//All Dump relays open  ******
IF (LCP.Section[1].Peak.DumpRelay1_close = FALSE AND
	LCP.Section[1].Peak.DumpRelay2_close = FALSE AND
	LCP.Section[1].Sust.DumpRelay1_close = FALSE AND
	LCP.Section[1].Sust.DumpRelay2_close = FALSE AND
	LCP.Section[2].Peak.DumpRelay1_close = FALSE AND
	LCP.Section[2].Peak.DumpRelay2_close = FALSE AND
	LCP.Section[2].Sust.DumpRelay1_close = FALSE AND
	LCP.Section[2].Sust.DumpRelay2_close = FALSE AND
	LCP.Section[3].Peak.DumpRelay1_close = FALSE AND
	LCP.Section[3].Peak.DumpRelay2_close = FALSE AND
	LCP.Section[3].Sust.DumpRelay1_close = FALSE AND
	LCP.Section[3].Sust.DumpRelay2_close = FALSE AND
	
	LCP.Section[4].Form.DumpRelay1_close = FALSE AND
	LCP.Section[4].Form.DumpRelay2_close = FALSE AND						
	LCP.Section[4].Form.PreFormDumpRly_close = FALSE AND
	LCP.Section[4].Form.FormTrigDumpRly1_close = FALSE AND
	LCP.Section[4].Form.PreFormTrigDumpRly1_close = FALSE) OR HMI_DB.AllDumpRelaysOpenBP = TRUE //admin bypass 
	THEN
		Permissives_DB.AllDumpRelaysOpen := TRUE;
	ELSE
		Permissives_DB.AllDumpRelaysOpen := FALSE;
END_IF;
//check for cap voltage for fully discharged
FOR i := 1 TO 3 BY 1 DO
	//peak
	FOR k := 1 TO 10 BY 1 DO
		IF LCP.Section[i].Peak.Cap[k].voltageFeedback <= 10 THEN 
			LCP.Section[i].Peak.Cap[k].CapDischaged := TRUE;
			ELSE
				LCP.Section[i].Peak.Cap[k].CapDischaged := FALSE;
		END_IF;
		//check for cap fully charged*************************
		IF LCP.Section[i].Peak.Cap[k].voltageFeedback >= Setpoints.TDKLoad[i].RequiredChargedV THEN 
			LCP.Section[i].Peak.Cap[k].CapfullyCharged := TRUE;
			ELSE
				LCP.Section[i].Peak.Cap[k].CapfullyCharged := FALSE;
		END_IF;
	END_FOR;
	//sus
	IF LCP.Section[i].Sust.Cap[1].voltageFeedback <= 10 THEN
		LCP.Section[i].Sust.Cap[1].CapDischaged := TRUE;
		ELSE
			LCP.Section[i].Sust.Cap[1].CapDischaged := FALSE;
	END_IF;
	//check fo cap fully charged
	IF LCP.Section[i].Sust.Cap[1].voltageFeedback >= Setpoints.TDKLoad[i+3].RequiredChargedV THEN
		LCP.Section[i].Sust.Cap[1].CapfullyCharged := TRUE;
		ELSE
			LCP.Section[i].Sust.Cap[1].CapfullyCharged := FALSE;
	END_IF;
	
	IF LCP.Section[i].Sust.Cap[2].voltageFeedback <= 10 THEN
		LCP.Section[i].Sust.Cap[2].CapDischaged := TRUE;
		ELSE
			LCP.Section[i].Sust.Cap[2].CapDischaged := FALSE;
	END_IF;
	//check for cap fully charged
	IF LCP.Section[i].Sust.Cap[2].voltageFeedback >= Setpoints.TDKLoad[i+3].RequiredChargedV THEN
		LCP.Section[i].Sust.Cap[2].CapfullyCharged := TRUE;
		ELSE
			LCP.Section[i].Sust.Cap[2].CapfullyCharged := FALSE;
	END_IF;
END_FOR;
// form
FOR m := 1 TO 12 BY 1 DO
	IF LCP.Section[4].Form.Cap[m].voltageFeedback <= 10 THEN
		LCP.Section[4].Form.Cap[m].CapDischaged := TRUE;
		ELSE
			LCP.Section[4].Form.Cap[m].CapDischaged := FALSE;
	END_IF;
END_FOR;

//check for cap fully charged
FOR n := 1 TO 6 BY 1 DO 
	IF LCP.Section[4].Form.Cap[n].voltageFeedback >= Setpoints.TDKLoad[7].RequiredChargedV THEN
		LCP.Section[4].Form.Cap[n].CapfullyCharged := TRUE;
		ELSE
			LCP.Section[4].Form.Cap[n].CapfullyCharged := FALSE;
	END_IF;		
END_FOR

FOR p := 7 TO 12 BY 1 DO 
	IF LCP.Section[4].Form.Cap[p].voltageFeedback >= Setpoints.TDKLoad[8].RequiredChargedV THEN
		LCP.Section[4].Form.Cap[p].CapfullyCharged := TRUE;
		ELSE
			LCP.Section[4].Form.Cap[p].CapfullyCharged := FALSE;
	END_IF;		
END_FOR

//preform
IF LCP.Section[4].PreFormCapVoltageFeedback <= 10 THEN
	LCP.Section[4].PreFormCapDischarged := TRUE;
	ELSE
		LCP.Section[4].PreFormCapDischarged := FALSE;
END_IF

//preform
IF LCP.Section[4].PreFormCapVoltageFeedback >= Setpoints.GLSLoad.RequiredChargedV THEN
	LCP.Section[4].PreFormCapFullyChaged := TRUE;
	ELSE
		LCP.Section[4].PreFormCapFullyChaged := FALSE;
END_IF


//all caps discharge condition
FOR i := 1 TO 3 BY 1 DO
	IF LCP.Section[i].Peak.Cap[1].CapDischaged = TRUE AND
		LCP.Section[i].Peak.Cap[2].CapDischaged = TRUE AND
		LCP.Section[i].Peak.Cap[3].CapDischaged = TRUE AND
		LCP.Section[i].Peak.Cap[4].CapDischaged = TRUE AND
		LCP.Section[i].Peak.Cap[5].CapDischaged = TRUE AND
		LCP.Section[i].Peak.Cap[6].CapDischaged = TRUE AND
		LCP.Section[i].Peak.Cap[7].CapDischaged = TRUE AND
		LCP.Section[i].Peak.Cap[8].CapDischaged = TRUE AND
		LCP.Section[i].Peak.Cap[9].CapDischaged = TRUE AND
		LCP.Section[i].Peak.Cap[10].CapDischaged = TRUE AND
		LCP.Section[i].Sust.Cap[1].CapDischaged = TRUE AND
		LCP.Section[i].Sust.Cap[2].CapDischaged = TRUE
		THEN
			LCP.Section[i].AllCapsDischarged := TRUE; 
		ELSE
			LCP.Section[i].AllCapsDischarged := FALSE; 
	END_IF;
	
	//all caps fully charged 
	IF LCP.Section[i].Peak.Cap[1].CapFullyCharged = TRUE AND
		LCP.Section[i].Peak.Cap[2].CapFullyCharged = TRUE AND
		LCP.Section[i].Peak.Cap[3].CapFullyCharged = TRUE AND
		LCP.Section[i].Peak.Cap[4].CapFullyCharged = TRUE AND
		LCP.Section[i].Peak.Cap[5].CapFullyCharged = TRUE AND
		LCP.Section[i].Peak.Cap[6].CapFullyCharged = TRUE AND
		LCP.Section[i].Peak.Cap[7].CapFullyCharged = TRUE AND
		LCP.Section[i].Peak.Cap[8].CapFullyCharged = TRUE AND
		LCP.Section[i].Peak.Cap[9].CapFullyCharged = TRUE AND
		LCP.Section[i].Peak.Cap[10].CapFullyCharged = TRUE AND
		LCP.Section[i].Sust.Cap[1].CapFullyCharged = TRUE AND
		LCP.Section[i].Sust.Cap[2].CapFullyCharged = TRUE
		THEN
			LCP.Section[i].AllCapsFullyCharged := TRUE;
		ELSE
			LCP.Section[i].AllCapsFullyCharged := FALSE;
	END_IF
END_FOR
//form caps 
IF LCP.Section[4].Form.Cap[1].CapDischaged = TRUE AND
	LCP.Section[4].Form.Cap[2].CapDischaged = TRUE AND
	LCP.Section[4].Form.Cap[3].CapDischaged = TRUE AND
	LCP.Section[4].Form.Cap[4].CapDischaged = TRUE AND
	LCP.Section[4].Form.Cap[5].CapDischaged = TRUE AND
	LCP.Section[4].Form.Cap[6].CapDischaged = TRUE AND
	LCP.Section[4].Form.Cap[7].CapDischaged = TRUE AND
	LCP.Section[4].Form.Cap[8].CapDischaged = TRUE AND
	LCP.Section[4].Form.Cap[9].CapDischaged = TRUE AND
	LCP.Section[4].Form.Cap[10].CapDischaged = TRUE AND
	LCP.Section[4].Form.Cap[11].CapDischaged = TRUE AND
	LCP.Section[4].Form.Cap[12].CapDischaged = TRUE AND 
	LCP.Section[4].PreFormCapDischarged = TRUE
	THEN 
		LCP.Section[4].AllCapsDischarged := TRUE;
	ELSE
		LCP.Section[4].AllCapsDischarged := FALSE;	
END_IF
//checking for caps fully charged
IF LCP.Section[4].Form.Cap[1].CapFullyCharged = TRUE AND
	LCP.Section[4].Form.Cap[2].CapFullyCharged = TRUE AND
	LCP.Section[4].Form.Cap[3].CapFullyCharged = TRUE AND
	LCP.Section[4].Form.Cap[4].CapFullyCharged = TRUE AND
	LCP.Section[4].Form.Cap[5].CapFullyCharged = TRUE AND
	LCP.Section[4].Form.Cap[6].CapFullyCharged = TRUE AND
	LCP.Section[4].Form.Cap[7].CapFullyCharged = TRUE AND
	LCP.Section[4].Form.Cap[8].CapFullyCharged = TRUE AND
	LCP.Section[4].Form.Cap[9].CapFullyCharged = TRUE AND
	LCP.Section[4].Form.Cap[10].CapFullyCharged = TRUE AND
	LCP.Section[4].Form.Cap[11].CapFullyCharged = TRUE AND
	LCP.Section[4].Form.Cap[12].CapFullyCharged = TRUE AND
	LCP.Section[4].PreFormCapFullyChaged = TRUE
	THEN
		LCP.Section[4].AllCapsFullyCharged := TRUE;
	ELSE
		LCP.Section[4].AllCapsFullyCharged := FALSE;
END_IF

//all capps fully charged
IF LCP.Section[1].AllCapsFullyCharged = TRUE AND
	LCP.Section[2].AllCapsFullyCharged = TRUE AND
	LCP.Section[3].AllCapsFullyCharged = TRUE AND
	LCP.Section[4].AllCapsFullyCharged = TRUE 
	THEN
		Permissives_DB.AllSectCapsFullyCharged := TRUE;
	ELSE
		Permissives_DB.AllSectCapsFullyCharged := FALSE;
END_IF

IF LCP.Section[1].AllCapsDischarged = TRUE AND
	LCP.Section[2].AllCapsDischarged = TRUE AND
	LCP.Section[3].AllCapsDischarged = TRUE AND
	LCP.Section[4].AllCapsDischarged = TRUE 
	THEN 
		Permissives_DB.AllSectCapsDischarged := TRUE;
	ELSE
		Permissives_DB.AllSectCapsDischarged := FALSE;
END_IF


//no loss in interlock pneumatic pressure

IF (LCP.Section[1].LossPneumaticPressure = FALSE AND
	LCP.Section[2].LossPneumaticPressure = FALSE AND
	LCP.Section[3].LossPneumaticPressure = FALSE AND
	LCP.Section[4].LossPneumaticPressure = FALSE) OR HMI_DB.InterlockPressureLossBP = TRUE 
	THEN
		Permissives_DB.NoInterlockPressureLoss := TRUE;
		ELSE
			Permissives_DB.NoInterlockPressureLoss := FALSE;
END_IF;
	
IF (Permissives_DB.NoShortingUnknowns = TRUE AND
	Trips_DB.AllDCpsuOK = TRUE AND
	Trips_DB.CageEStopCircuitBroken = FALSE AND
	Trips_DB.AnyChargerOverTemp = FALSE AND
	Trips_DB.AnyEstopPressed = FALSE AND
	Trips_DB.AnyChargerInterlockOpen = FALSE AND
	Permissives_DB.NoInterlockPressureLoss = TRUE) OR HMI_DB.SafetyOKBP = TRUE // admin bypass 
	THEN
		Permissives_DB.SafetyOK := TRUE;
		ELSE
			Permissives_DB.SafetyOK := FALSE;
END_IF;

IF i > 3 THEN
	i := 1;
END_IF;

IF j > 8 THEN
	j := 1;
END_IF;

IF k > 10 THEN
	k := 1;
END_IF;

IF m > 12 THEN
	m := 1;
END_IF;

IF n > 6 THEN
	n := 1;
END_IF;

IF p > 12 THEN
	p := 7;
END_IF;

END_PROGRAM

// ---- POUs/Trips.TcPOU
PROGRAM Trips
VAR
	bTest							: BOOL;
	//delay2s : Delay2s;
	evtLogger						: FB_TcEventLogger;
	
	ACintLockRlyFaultDelay_PT		: TIME := T#2S;
	DumpRlyFaultDelay_PT			: TIME := T#2S;
	//DumpRly2FaultDelay_PT			: TIME := T#2S;
	ChrgRlyFaultDelay_PT			: TIME := T#1S;
	
	LiftMachineGNDFaultTON			: TON;
	LiftMachineGNDFaultPT			: TIME := T#2000MS;
	
	GeneralFaultDelayPT				: TIME := T#500MS;
	
	stControl						: ST_Control;
	
	i : INT := 1;  //charger 1-8
	j : INT := 1; //section 1-3
	k : INT := 1; //section 1-4, might not need 
END_VAR


//MCP Input Trips
IF MCP_IO.MasterStopPB_Pressed = TRUE THEN
	Trips_DB.MasterStopPBPressed := TRUE;	
END_IF;

IF MCP_IO.CageEstopCircuitOK = FALSE THEN
	Trips_DB.CageEStopCircuitBroken := TRUE; 
END_IF;

IF MCP_IO.RemoteModeSelected = FALSE THEN
	Trips_DB.LocalModeSelected := TRUE; //may not be a trip
	ELSE
		Trips_DB.LocalModeSelected := FALSE;
END_IF;

IF MCP_IO.PSU1_DCOK = FALSE THEN
	Trips_DB.MCPLossDCpower := TRUE; 
END_IF;

IF (MCP_IO.LiftMachineGND = TRUE AND MCP_IO.MachineGNDrlyOpen = FALSE) OR 
	(MCP_IO.LiftMachineGND = FALSE AND MCP_IO.MachineGNDrlyOpen = TRUE)
	THEN
		//delay
		LiftMachineGNDFaultTON (IN := TRUE, PT := LiftMachineGNDFaultPT);
		IF LiftMachineGNDFaultTON.Q = TRUE THEN
			Trips_DB.MachineGNDrlyFailed := TRUE;
			LiftMachineGNDFaultTON (IN := FALSE);
		END_IF
	ELSE
		LiftMachineGNDFaultTON (IN := FALSE);
END_IF

//FOR i := 1 TO 8 BY 1 DO
FOR i := 1 TO 3 BY 1 DO	//only has 3 chargers in this version
	//check for loss inhibit

	IF (MCP_IO.Charger[i].inhibit = TRUE AND MCP_IO.Charger[i].inhibited = FALSE) OR 
		(MCP_IO.Charger[i].inhibit = FALSE AND MCP_IO.Charger[i].inhibited = TRUE)
		THEN
			MCP_IO.Charger[i].LossInhibitTON (IN := TRUE, PT := GeneralFaultDelayPT);
			IF MCP_IO.Charger[i].LossInhibitTON.Q = TRUE THEN 
				MCP_IO.Charger[i].LossInhibit := TRUE; //for alarms and not an actual trip
				MCP_IO.Charger[i].LossInhibitTON (IN := FALSE);
			END_IF
		ELSE
			MCP_IO.Charger[i].LossInhibit := FALSE;
			MCP_IO.Charger[i].LossInhibitTON (IN := FALSE);
	END_IF
	//check for loss HV on signal
	IF MCP_IO.Charger[i].HV_ON = TRUE AND MCP_IO.Charger[i].HV_isON = FALSE 
		THEN
			MCP_IO.Charger[i].LossHVON_TON (IN := TRUE, PT := GeneralFaultDelayPT);
			IF MCP_IO.Charger[i].LossHVON_TON.Q = TRUE THEN
				MCP_IO.Charger[i].LossHVON := TRUE; //for alarms and not an actual trip
				MCP_IO.Charger[i].LossHVON_TON (IN := FALSE);
			END_IF
		ELSE
			MCP_IO.Charger[i].LossHVON := FALSE;
			MCP_IO.Charger[i].LossHVON_TON (IN := FALSE);
	END_IF
	//any loss inhibit signal and hv on signal
	IF MCP_IO.Charger[i].LossInhibit = TRUE THEN 
		Trips_DB.AnyLossInhibitSignal := TRUE;
	END_IF

END_FOR;

IF ((MCP_IO.Charger[1].LossHVON = TRUE AND Recipe.PeakSupplyEN = TRUE) OR
	(MCP_IO.Charger[2].LossHVON = TRUE AND Recipe.PeakSupplyEN = TRUE) OR
	(MCP_IO.Charger[3].LossHVON = TRUE AND Recipe.PeakSupplyEN = TRUE) (*OR
	(MCP_IO.Charger[4].LossHVON = TRUE AND Recipe.SustSupplyEN = TRUE) OR
	(MCP_IO.Charger[5].LossHVON = TRUE AND Recipe.SustSupplyEN = TRUE) OR
	(MCP_IO.Charger[6].LossHVON = TRUE AND Recipe.SustSupplyEN = TRUE) OR
	(MCP_IO.Charger[7].LossHVON = TRUE AND Recipe.FormSupplyEN = TRUE) OR
	(MCP_IO.Charger[8].LossHVON = TRUE AND Recipe.FormSupplyEN = TRUE)*)) AND HMI_DB.LossHVsignalBP = FALSE 
THEN
	Trips_DB.AnyLossHVONsignal := TRUE;
END_IF


// mapping pnumatic and dc power to trips
FOR k := 1 TO 4 BY 1 DO
	Trips_DB.Section[k].LossPneumaticPressure := LCP.Section[k].LossPneumaticPressure;
	Trips_DB.Section[k].LossDCPower := NOT LCP.Section[k].PSU1_DCOK;
END_FOR;


//any charge relay fail
IF Trips_DB.Section[1].Peak.ChargeRelay1_Failed = TRUE OR
	Trips_DB.Section[1].Peak.ChargeRelay2_Failed = TRUE OR
	Trips_DB.Section[1].Sust.ChargeRelay1_Failed = TRUE OR
	Trips_DB.Section[1].Sust.ChargeRelay2_Failed = TRUE OR
	Trips_DB.Section[2].Peak.ChargeRelay1_Failed = TRUE OR
	Trips_DB.Section[2].Peak.ChargeRelay2_Failed = TRUE OR
	Trips_DB.Section[2].Sust.ChargeRelay1_Failed = TRUE OR
	Trips_DB.Section[2].Sust.ChargeRelay2_Failed = TRUE OR
	Trips_DB.Section[3].Peak.ChargeRelay1_Failed = TRUE OR
	Trips_DB.Section[3].Peak.ChargeRelay2_Failed = TRUE OR
	Trips_DB.Section[3].Sust.ChargeRelay1_Failed = TRUE OR
	Trips_DB.Section[3].Sust.ChargeRelay2_Failed = TRUE OR
	Trips_DB.Section[4].Form.ChargeRelay1_Failed = TRUE OR 
	Trips_DB.Section[4].Form.ChargeRelay2_Failed = TRUE OR 
	Trips_DB.Section[4].Form.PreFormChrgRlyFailed = TRUE OR 
	Trips_DB.Section[4].Form.FormTrigChrgRlyFailed = TRUE OR
	Trips_DB.Section[4].Form.PreFormTrigChrgRlyFailed = TRUE		
	THEN 
		Trips_DB.AnyChargeRlyFail := TRUE;
	ELSE
		Trips_DB.AnyChargeRlyFail := FALSE;
END_IF;

//any dump relay fail
IF Trips_DB.Section[1].Peak.DumpRelay1_Failed = TRUE OR
	Trips_DB.Section[1].Peak.DumpRelay2_Failed = TRUE OR
	Trips_DB.Section[1].Sust.DumpRelay1_Failed = TRUE OR
	Trips_DB.Section[1].Sust.DumpRelay2_Failed = TRUE OR
	Trips_DB.Section[2].Peak.DumpRelay1_Failed = TRUE OR
	Trips_DB.Section[2].Peak.DumpRelay2_Failed = TRUE OR
	Trips_DB.Section[2].Sust.DumpRelay1_Failed = TRUE OR
	Trips_DB.Section[2].Sust.DumpRelay2_Failed = TRUE OR
	Trips_DB.Section[3].Peak.DumpRelay1_Failed = TRUE OR
	Trips_DB.Section[3].Peak.DumpRelay2_Failed = TRUE OR
	Trips_DB.Section[3].Sust.DumpRelay1_Failed = TRUE OR
	Trips_DB.Section[3].Sust.DumpRelay2_Failed = TRUE OR
	Trips_DB.Section[4].Form.DumpRelay1_Failed = TRUE OR 
	Trips_DB.Section[4].Form.DumpRelay2_Failed = TRUE OR 
	Trips_DB.Section[4].Form.PreFormDumpRlyFailed = TRUE OR 
	Trips_DB.Section[4].Form.FormTrigDumpRly1Failed = TRUE OR
	Trips_DB.Section[4].Form.PreFormTrigDumpRly1Failed = TRUE		
	THEN 
		Trips_DB.AnyDumpRlyFail := TRUE;
	ELSE
		Trips_DB.AnyDumpRlyFail := FALSE;
END_IF;

//if relays failed, chargers faulted, loss pneumatic pressure, or loss dc power then 
//Trips_DB.Section[j].SystemTripped := TRUE;

//system trip 
//section 1-3
FOR j := 1 TO 3 BY 1 DO
	IF Trips_DB.Section[j].LossDCPower = TRUE OR 
		Trips_DB.Section[j].LossPneumaticPressure = TRUE OR
		Trips_DB.Section[j].Peak.ChargeRelay1_Failed = TRUE OR
		Trips_DB.Section[j].Peak.ChargeRelay2_Failed = TRUE OR
		Trips_DB.Section[j].Peak.DumpRelay1_Failed = TRUE OR
		Trips_DB.Section[j].Peak.DumpRelay2_Failed = TRUE OR
		Trips_DB.Section[j].Sust.ChargeRelay1_Failed = TRUE OR
		Trips_DB.Section[j].Sust.ChargeRelay2_Failed = TRUE OR
		Trips_DB.Section[j].Sust.DumpRelay1_Failed = TRUE OR
		Trips_DB.Section[j].Sust.DumpRelay2_Failed = TRUE OR
		// shorted when not supposed to ?
		LCP.Section[j].Peak.ShortContact1unknown = TRUE OR // might need to  test it.  
		LCP.Section[j].Peak.ShortContact2unknown = TRUE 
		THEN
			Trips_DB.Section[j].SystemTripped := TRUE;
	END_IF;
END_FOR;

//formation
IF Trips_DB.Section[4].LossDCPower = TRUE OR 
	Trips_DB.Section[4].LossPneumaticPressure = TRUE OR
	Trips_DB.Section[4].Form.ChargeRelay1_Failed = TRUE OR
	Trips_DB.Section[4].Form.ChargeRelay2_Failed = TRUE OR
	Trips_DB.Section[4].Form.DumpRelay1_Failed = TRUE OR
	Trips_DB.Section[4].Form.DumpRelay2_Failed = TRUE OR
	Trips_DB.Section[4].Form.PreFormChrgRlyFailed = TRUE OR
	Trips_DB.Section[4].Form.FormTrigChrgRlyFailed = TRUE OR
	Trips_DB.Section[4].Form.PreFormTrigChrgRlyFailed = TRUE OR
	Trips_DB.Section[4].Form.PreFormDumpRlyFailed = TRUE OR
	Trips_DB.Section[4].Form.FormTrigDumpRly1Failed = TRUE OR
	Trips_DB.Section[4].Form.PreFormTrigDumpRly1Failed = TRUE OR 
	LCP.Section[4].Form.ShortContact1unknown = TRUE OR //might need to remove, might be too sensitive
	LCP.Section[4].Form.ShortContact2unknown = TRUE OR 
	LCP.Section[4].Form.FormTrigShortContactUnknown = TRUE OR 
	LCP.Section[4].Form.PreFormTrigShortContactUnknown = TRUE
	THEN
		Trips_DB.Section[4].SystemTripped := TRUE;
END_IF;


//Charger faults
//FOR i := 1 TO 8 BY 1 DO
FOR i := 1 TO 3 BY 1 DO
	//OVERTEMP 
	IF MCP_IO.Charger[i].OverTemp = TRUE THEN
		Trips_DB.AnyChargerOverTemp := TRUE;  
	END_IF;
	//Load faults
	IF MCP_IO.Charger[i].LoadFaulted = TRUE THEN
		Trips_DB.AnyChargerLoadFault := TRUE;  
	END_IF;
	//Interlock Open
	IF MCP_IO.Charger[i].InterlockOpen = TRUE THEN
		Trips_DB.AnyChargerInterlockOpen := TRUE;  
	END_IF;
	
END_FOR;

//Charger summary faults
//FOR i := 1 TO 8 BY 1 DO
FOR i := 1 TO 3 BY 1 DO
	IF MCP_IO.Charger[i].SummaryFaulted = TRUE THEN
		Trips_DB.AnyChargerFaulted := TRUE;  
	END_IF;
END_FOR;

//MCP trip
IF Trips_DB.AnyChargerFaulted = TRUE OR 
	Trips_DB.MasterStopPBPressed = TRUE OR
	Trips_DB.CageEStopCircuitBroken = TRUE OR
	Trips_DB.MCPLossDCpower = TRUE 
	THEN
		Trips_DB.MCPsystemTripped := TRUE;
END_IF


//*******************E-Stop Trips
IF MCP_IO.MasterStopPB_Pressed = TRUE OR MCP_IO.CageEstopCircuitOK THEN
	Trips_DB.AnyEstopPressed := TRUE;  
END_IF;	

//*********************DC PSU
IF (MCP_IO.PSU1_DCOK = TRUE AND 
	LCP.Section[1].PSU1_DCOK = TRUE AND
	LCP.Section[2].PSU1_DCOK = TRUE AND
	LCP.Section[3].PSU1_DCOK = TRUE AND
	LCP.Section[4].PSU1_DCOK = TRUE) OR HMI_DB.AlldcPSUokBP = TRUE //admin bypass 
	THEN
		TRIPS_DB.AllDCpsuOK := TRUE;
	ELSE 
		TRIPS_DB.AllDCpsuOK := FALSE;
END_IF;

//Relay faults***************************************
//section 1 - 3
FOR j := 1 TO 3 BY 1 DO
	//Peak Charge rly1
		//fail to close
	IF LCP.Section[j].Peak.CloseChargeRelay1 = TRUE AND LCP.Section[j].Peak.ChargeRelay1_close = FALSE THEN 
		//start timer
		Trips_DB.Section[j].Peak.ChrgRly1FaultDelay_TON (IN:= TRUE, PT := ChrgRlyFaultDelay_PT);
		
		IF Trips_DB.Section[j].Peak.ChrgRly1FaultDelay_TON.Q = TRUE THEN 
			Trips_DB.Section[j].Peak.ChargeRelay1_FailtoClose := TRUE; 
			Trips_DB.Section[j].Peak.ChrgRly1FaultDelay_TON (IN:= FALSE);
		END_IF;
	ELSE
		Trips_DB.Section[j].Peak.ChrgRly1FaultDelay_TON (IN:= FALSE);
	END_IF;

		//fail to open
	IF LCP.Section[j].Peak.CloseChargeRelay1 = FALSE AND LCP.Section[j].Peak.ChargeRelay1_close = TRUE THEN 
		//start timer
		Trips_DB.Section[j].Peak.ChrgRly1FaultDelay_TON (IN:= TRUE, PT := ChrgRlyFaultDelay_PT);
		
		IF Trips_DB.Section[j].Peak.ChrgRly1FaultDelay_TON.Q = TRUE THEN 
			Trips_DB.Section[j].Peak.ChargeRelay1_FailtoOpen := TRUE; 
			Trips_DB.Section[j].Peak.ChrgRly1FaultDelay_TON (IN:= FALSE);
		END_IF;
	ELSE
		Trips_DB.Section[j].Peak.ChrgRly1FaultDelay_TON (IN:= FALSE);
	END_IF;

	//Peak Charge rly2	
		//fail to close
	IF LCP.Section[j].Peak.CloseChargeRelay2 = TRUE AND LCP.Section[j].Peak.ChargeRelay2_close = FALSE THEN 
		//start timer
		Trips_DB.Section[j].Peak.ChrgRly2FaultDelay_TON (IN:= TRUE, PT := ChrgRlyFaultDelay_PT);
		
		IF Trips_DB.Section[j].Peak.ChrgRly2FaultDelay_TON.Q = TRUE THEN 
			Trips_DB.Section[j].Peak.ChargeRelay2_FailtoClose := TRUE; 
			Trips_DB.Section[j].Peak.ChrgRly2FaultDelay_TON (IN:= FALSE);
		END_IF;
	ELSE
		Trips_DB.Section[j].Peak.ChrgRly2FaultDelay_TON (IN:= FALSE);
	END_IF;
	
		//fail to open
	IF LCP.Section[j].Peak.CloseChargeRelay2 = FALSE AND LCP.Section[j].Peak.ChargeRelay2_close = TRUE THEN 
		//start timer
		Trips_DB.Section[j].Peak.ChrgRly2FaultDelay_TON (IN:= TRUE, PT := ChrgRlyFaultDelay_PT);
		
		IF Trips_DB.Section[j].Peak.ChrgRly2FaultDelay_TON.Q = TRUE THEN 
			Trips_DB.Section[j].Peak.ChargeRelay2_FailtoOpen := TRUE; 
			Trips_DB.Section[j].Peak.ChrgRly2FaultDelay_TON (IN:= FALSE);
		END_IF;
	ELSE
		Trips_DB.Section[j].Peak.ChrgRly2FaultDelay_TON (IN:= FALSE);
	END_IF;

	//Peak dump rly1
		//fail to open
	IF LCP.Section[j].Peak.OpenDumpRelay1 = TRUE AND LCP.Section[j].Peak.DumpRelay1_close = TRUE THEN 
		//start timer
		Trips_DB.Section[j].Peak.DumpRly1FaultDelay_TON (IN := TRUE, PT := DumpRlyFaultDelay_PT);

		IF Trips_DB.Section[j].Peak.DumpRly1FaultDelay_TON.Q = TRUE THEN 
			Trips_DB.Section[j].Peak.DumpRelay1_FailtoOpen := TRUE; 
			Trips_DB.Section[j].Peak.DumpRly1FaultDelay_TON (IN:= FALSE);
		END_IF; 
	ELSE
		Trips_DB.Section[j].Peak.DumpRly1FaultDelay_TON (IN:= FALSE);
	END_IF;

		//fail to close
	IF LCP.Section[j].Peak.OpenDumpRelay1 = FALSE AND LCP.Section[j].Peak.DumpRelay1_close = FALSE THEN 
		//start timer
		Trips_DB.Section[j].Peak.DumpRly1FaultDelay_TON (IN := TRUE, PT := DumpRlyFaultDelay_PT); 
		
		IF Trips_DB.Section[j].Peak.DumpRly1FaultDelay_TON.Q = TRUE THEN 
			Trips_DB.Section[j].Peak.DumpRelay1_FailtoClose := TRUE;
			Trips_DB.Section[j].Peak.DumpRly1FaultDelay_TON (IN:= FALSE);
		END_IF;
	ELSE
		Trips_DB.Section[j].Peak.DumpRly1FaultDelay_TON (IN:= FALSE);
	END_IF;

	//Peak dump rly2
		//fail to open
	IF LCP.Section[j].Peak.OpenDumpRelay2 = TRUE AND LCP.Section[j].Peak.DumpRelay2_close = TRUE THEN 
		//start timer
		Trips_DB.Section[j].Peak.DumpRly2FaultDelay_TON (IN := TRUE, PT := DumpRlyFaultDelay_PT); 
		
		IF Trips_DB.Section[j].Peak.DumpRly2FaultDelay_TON.Q = TRUE THEN 
			Trips_DB.Section[j].Peak.DumpRelay2_FailtoOpen := TRUE; 
			Trips_DB.Section[j].Peak.DumpRly2FaultDelay_TON (IN:= FALSE);
		END_IF;
	ELSE
		Trips_DB.Section[j].Peak.DumpRly2FaultDelay_TON (IN:= FALSE);
	END_IF;

		//fail to close
	IF LCP.Section[j].Peak.OpenDumpRelay2 = FALSE AND LCP.Section[j].Peak.DumpRelay2_close = FALSE THEN 
		//start timer
		Trips_DB.Section[j].Peak.DumpRly2FaultDelay_TON (IN := TRUE, PT := DumpRlyFaultDelay_PT); 
		IF Trips_DB.Section[j].Peak.DumpRly2FaultDelay_TON.Q = TRUE THEN 
			Trips_DB.Section[j].Peak.DumpRelay2_FailtoClose := TRUE; 
			
		END_IF;
	ELSE
		Trips_DB.Section[j].Peak.DumpRly2FaultDelay_TON (IN:= FALSE);
	END_IF;
//*************************************************************************************************

//Sust Charge rly1
		//fail to close
	IF LCP.Section[j].Sust.CloseChargeRelay1 = TRUE AND LCP.Section[j].Sust.ChargeRelay1_close = FALSE THEN 
		//start timer
		Trips_DB.Section[j].Sust.ChrgRly1FaultDelay_TON (IN:= TRUE, PT := ChrgRlyFaultDelay_PT);
		
		IF Trips_DB.Section[j].Sust.ChrgRly1FaultDelay_TON.Q = TRUE THEN 
			Trips_DB.Section[j].Sust.ChargeRelay1_FailtoClose := TRUE; 
			Trips_DB.Section[j].Sust.ChrgRly1FaultDelay_TON (IN:= FALSE);
		END_IF;
	ELSE
		Trips_DB.Section[j].Sust.ChrgRly1FaultDelay_TON (IN:= FALSE);	
	END_IF;

		//fail to open
	IF LCP.Section[j].Sust.CloseChargeRelay1 = FALSE AND LCP.Section[j].Sust.ChargeRelay1_close = TRUE THEN 
		//start timer
		Trips_DB.Section[j].Sust.ChrgRly1FaultDelay_TON (IN:= TRUE, PT := ChrgRlyFaultDelay_PT);
		
		IF Trips_DB.Section[j].Sust.ChrgRly1FaultDelay_TON.Q = TRUE THEN 
			Trips_DB.Section[j].Sust.ChargeRelay1_FailtoOpen := TRUE; 
			Trips_DB.Section[j].Sust.ChrgRly1FaultDelay_TON (IN:= FALSE);
		END_IF;
	ELSE
		Trips_DB.Section[j].Sust.ChrgRly1FaultDelay_TON (IN:= FALSE);
	END_IF;

	//Sust Charge rly2	
		//fail to close
	IF LCP.Section[j].Sust.CloseChargeRelay2 = TRUE AND LCP.Section[j].Sust.ChargeRelay2_close = FALSE THEN 
		//start timer
		Trips_DB.Section[j].Sust.ChrgRly2FaultDelay_TON (IN:= TRUE, PT := ChrgRlyFaultDelay_PT);
		
		IF Trips_DB.Section[j].Sust.ChrgRly2FaultDelay_TON.Q = TRUE THEN 
			Trips_DB.Section[j].Sust.ChargeRelay2_FailtoClose := TRUE;
			Trips_DB.Section[j].Sust.ChrgRly2FaultDelay_TON (IN:= FALSE);
		END_IF;
	ELSE
		Trips_DB.Section[j].Sust.ChrgRly2FaultDelay_TON (IN:= FALSE);
	END_IF;
	
		//fail to open
	IF LCP.Section[j].Sust.CloseChargeRelay2 = FALSE AND LCP.Section[j].Sust.ChargeRelay2_close = TRUE THEN 
		//start timer
		Trips_DB.Section[j].Sust.ChrgRly2FaultDelay_TON (IN:= TRUE, PT := ChrgRlyFaultDelay_PT);
		
		IF Trips_DB.Section[j].Sust.ChrgRly2FaultDelay_TON.Q = TRUE THEN 
			Trips_DB.Section[j].Sust.ChargeRelay2_FailtoOpen := TRUE; 
			Trips_DB.Section[j].Sust.ChrgRly2FaultDelay_TON (IN:= FALSE);
		END_IF;
	ELSE
		Trips_DB.Section[j].Sust.ChrgRly2FaultDelay_TON (IN:= FALSE);
	END_IF;

	//Sust dump rly1
		//fail to open
	IF LCP.Section[j].Sust.OpenDumpRelay1 = TRUE AND LCP.Section[j].Sust.DumpRelay1_close = TRUE THEN 
		//start timer
		Trips_DB.Section[j].Sust.DumpRly1FaultDelay_TON (IN := TRUE, PT := DumpRlyFaultDelay_PT);

		IF Trips_DB.Section[j].Sust.DumpRly1FaultDelay_TON.Q = TRUE THEN 
			Trips_DB.Section[j].Sust.DumpRelay1_FailtoOpen := TRUE; 
			Trips_DB.Section[j].Sust.DumpRly1FaultDelay_TON (IN:= FALSE);
		END_IF; 
	ELSE
		Trips_DB.Section[j].Sust.DumpRly1FaultDelay_TON (IN:= FALSE);
	END_IF;

		//fail to close
	IF LCP.Section[j].Sust.OpenDumpRelay1 = FALSE AND LCP.Section[j].Sust.DumpRelay1_close = FALSE THEN 
		//start timer
		Trips_DB.Section[j].Sust.DumpRly1FaultDelay_TON (IN := TRUE, PT := DumpRlyFaultDelay_PT); 
		
		IF Trips_DB.Section[j].Sust.DumpRly1FaultDelay_TON.Q = TRUE THEN 
			Trips_DB.Section[j].Sust.DumpRelay1_FailtoClose := TRUE; 
			Trips_DB.Section[j].Sust.DumpRly1FaultDelay_TON (IN:= FALSE);
		END_IF;
	ELSE
		Trips_DB.Section[j].Sust.DumpRly1FaultDelay_TON (IN:= FALSE);
	END_IF;

	//Sust dump rly2
		//fail to open
	IF LCP.Section[j].Sust.OpenDumpRelay2 = TRUE AND LCP.Section[j].Sust.DumpRelay2_close = TRUE THEN 
		//start timer
		Trips_DB.Section[j].Sust.DumpRly2FaultDelay_TON (IN := TRUE, PT := DumpRlyFaultDelay_PT); 
		
		IF Trips_DB.Section[j].Sust.DumpRly2FaultDelay_TON.Q = TRUE THEN 
			Trips_DB.Section[j].Sust.DumpRelay2_FailtoOpen := TRUE; 
			Trips_DB.Section[j].Sust.DumpRly2FaultDelay_TON (IN:= FALSE);
		END_IF;
	ELSE
		Trips_DB.Section[j].Sust.DumpRly2FaultDelay_TON (IN:= FALSE);
	END_IF;

		//fail to close
	IF LCP.Section[j].Sust.OpenDumpRelay2 = FALSE AND LCP.Section[j].Sust.DumpRelay2_close = FALSE THEN 
		//start timer
		Trips_DB.Section[j].Sust.DumpRly2FaultDelay_TON (IN := TRUE, PT := DumpRlyFaultDelay_PT); 
		IF Trips_DB.Section[j].Sust.DumpRly2FaultDelay_TON.Q = TRUE THEN 
			Trips_DB.Section[j].Sust.DumpRelay2_FailtoClose := TRUE; 
			Trips_DB.Section[j].Sust.DumpRly2FaultDelay_TON (IN:= FALSE);
		END_IF;
	ELSE
		Trips_DB.Section[j].Sust.DumpRly2FaultDelay_TON (IN:= FALSE);
	END_IF;
	
END_FOR;
//****************************************	
	
//Form Charge rly1
		//fail to close
IF LCP.Section[4].Form.CloseChargeRelay1 = TRUE AND LCP.Section[4].Form.ChargeRelay1_close = FALSE THEN 
		//start timer
		Trips_DB.Section[4].Form.ChrgRly1FaultDelay_TON (IN:= TRUE, PT := ChrgRlyFaultDelay_PT);
		
		IF Trips_DB.Section[4].Form.ChrgRly1FaultDelay_TON.Q = TRUE THEN 
			Trips_DB.Section[4].Form.ChargeRelay1_FailtoClose := TRUE; 
			Trips_DB.Section[4].Form.ChrgRly1FaultDelay_TON (IN:= FALSE);
		END_IF;
	ELSE
		Trips_DB.Section[4].Form.ChrgRly1FaultDelay_TON (IN:= FALSE);		
END_IF;

		//fail to open
IF LCP.Section[4].Form.CloseChargeRelay1 = FALSE AND LCP.Section[4].Form.ChargeRelay1_close = TRUE THEN 
		//start timer
		Trips_DB.Section[4].Form.ChrgRly1FaultDelay_TON (IN:= TRUE, PT := ChrgRlyFaultDelay_PT);
		
		IF Trips_DB.Section[4].Form.ChrgRly1FaultDelay_TON.Q = TRUE THEN 
			Trips_DB.Section[4].Form.ChargeRelay1_FailtoOpen := TRUE; 
			Trips_DB.Section[4].Form.ChrgRly1FaultDelay_TON (IN:= FALSE);
		END_IF;
	ELSE
		Trips_DB.Section[4].Form.ChrgRly1FaultDelay_TON (IN:= FALSE);
END_IF;

	//Form Charge rly2	
		//fail to close
IF LCP.Section[4].Form.CloseChargeRelay2 = TRUE AND LCP.Section[4].Form.ChargeRelay2_close = FALSE THEN 
		//start timer
		Trips_DB.Section[4].Form.ChrgRly2FaultDelay_TON (IN:= TRUE, PT := ChrgRlyFaultDelay_PT);
		
		IF Trips_DB.Section[4].Form.ChrgRly2FaultDelay_TON.Q = TRUE THEN 
			Trips_DB.Section[4].Form.ChargeRelay2_FailtoClose := TRUE; 
			Trips_DB.Section[4].Form.ChrgRly2FaultDelay_TON (IN:= FALSE);
		END_IF;
	ELSE
		Trips_DB.Section[4].Form.ChrgRly2FaultDelay_TON (IN:= FALSE);
END_IF;
	
		//fail to open
IF LCP.Section[4].Form.CloseChargeRelay2 = FALSE AND LCP.Section[4].Form.ChargeRelay2_close = TRUE THEN 
		//start timer
		Trips_DB.Section[4].Form.ChrgRly2FaultDelay_TON (IN:= TRUE, PT := ChrgRlyFaultDelay_PT);
		
		IF Trips_DB.Section[4].Form.ChrgRly2FaultDelay_TON.Q = TRUE THEN 
			Trips_DB.Section[4].Form.ChargeRelay2_FailtoOpen := TRUE; 
			Trips_DB.Section[4].Form.ChrgRly2FaultDelay_TON (IN:= FALSE);
		END_IF;
	ELSE
		Trips_DB.Section[4].Form.ChrgRly2FaultDelay_TON (IN:= FALSE);
END_IF;

	//Form dump rly1
		//fail to open
IF LCP.Section[4].Form.OpenDumpRelay1 = TRUE AND LCP.Section[4].Form.DumpRelay1_close = TRUE THEN 
		//start timer
		Trips_DB.Section[4].Form.DumpRly1FaultDelay_TON (IN := TRUE, PT := DumpRlyFaultDelay_PT);

		IF Trips_DB.Section[4].Form.DumpRly1FaultDelay_TON.Q = TRUE THEN 
			Trips_DB.Section[4].Form.DumpRelay1_FailtoOpen := TRUE; 
			Trips_DB.Section[4].Form.DumpRly1FaultDelay_TON (IN:= FALSE);
		END_IF; 
	ELSE
		Trips_DB.Section[4].Form.DumpRly1FaultDelay_TON (IN:= FALSE);
END_IF;

		//fail to close
IF LCP.Section[4].Form.OpenDumpRelay1 = FALSE AND LCP.Section[4].Form.DumpRelay1_close = FALSE THEN 
		//start timer
		Trips_DB.Section[4].Form.DumpRly1FaultDelay_TON (IN := TRUE, PT := DumpRlyFaultDelay_PT); 
		
		IF Trips_DB.Section[4].Form.DumpRly1FaultDelay_TON.Q = TRUE THEN 
			Trips_DB.Section[4].Form.DumpRelay1_FailtoClose := TRUE; 
			Trips_DB.Section[4].Form.DumpRly1FaultDelay_TON (IN:= FALSE);
		END_IF;
	ELSE
		Trips_DB.Section[4].Form.DumpRly1FaultDelay_TON (IN:= FALSE);
END_IF;

	//Form dump rly2
		//fail to open
IF LCP.Section[4].Form.OpenDumpRelay2 = TRUE AND LCP.Section[4].Form.DumpRelay2_close = TRUE THEN 
		//start timer
		Trips_DB.Section[4].Form.DumpRly2FaultDelay_TON (IN := TRUE, PT := DumpRlyFaultDelay_PT); 
		
		IF Trips_DB.Section[4].Form.DumpRly2FaultDelay_TON.Q = TRUE THEN 
			Trips_DB.Section[4].Form.DumpRelay2_FailtoOpen := TRUE; 
			Trips_DB.Section[4].Form.DumpRly2FaultDelay_TON (IN:= FALSE);
		END_IF;
	ELSE
		Trips_DB.Section[4].Form.DumpRly2FaultDelay_TON (IN:= FALSE);
END_IF;

		//fail to close
IF LCP.Section[4].Form.OpenDumpRelay2 = FALSE AND LCP.Section[4].Form.DumpRelay2_close = FALSE THEN 
		//start timer
		Trips_DB.Section[4].Form.DumpRly2FaultDelay_TON (IN := TRUE, PT := DumpRlyFaultDelay_PT); 
		IF Trips_DB.Section[4].Form.DumpRly2FaultDelay_TON.Q = TRUE THEN 
			Trips_DB.Section[4].Form.DumpRelay2_FailtoClose := TRUE; 
			Trips_DB.Section[4].Form.DumpRly2FaultDelay_TON (IN:= FALSE);
		END_IF;
	ELSE
		Trips_DB.Section[4].Form.DumpRly2FaultDelay_TON (IN:= FALSE);
END_IF;	

	//PreForm Charge rly
		//fail to close
IF (LCP.Section[4].Form.ClosePreFormChargeRly = TRUE AND LCP.Section[4].Form.PreFormChargeRly_close = FALSE) OR 
		(LCP.Section[4].Form.ClosePreFormChargeRly = FALSE AND LCP.Section[4].Form.PreFormChargeRly_close = TRUE) 
		THEN 
		//start timer
		Trips_DB.Section[4].Form.PreFormChrgRlyFaultDelay_TON (IN:= TRUE, PT := ChrgRlyFaultDelay_PT);
		
		IF Trips_DB.Section[4].Form.PreFormChrgRlyFaultDelay_TON.Q = TRUE THEN 
			Trips_DB.Section[4].Form.PreFormChrgRlyFailed := TRUE; 
			Trips_DB.Section[4].Form.PreFormChrgRlyFaultDelay_TON (IN:= FALSE);
		END_IF;
	ELSE
		Trips_DB.Section[4].Form.PreFormChrgRlyFaultDelay_TON (IN:= FALSE);
END_IF;

//form trigger charge 
		//fail to close
IF (LCP.Section[4].Form.CloseFormTrigChargeRly = TRUE AND LCP.Section[4].Form.FormTrigChargeRly_close = FALSE) OR 
		(LCP.Section[4].Form.CloseFormTrigChargeRly = FALSE AND LCP.Section[4].Form.FormTrigChargeRly_close = TRUE) 
		THEN 
		//start timer
		Trips_DB.Section[4].Form.FormTrigChrgRlyFaultDelay_TON (IN:= TRUE, PT := ChrgRlyFaultDelay_PT);
		
		IF Trips_DB.Section[4].Form.FormTrigChrgRlyFaultDelay_TON.Q = TRUE THEN 
			Trips_DB.Section[4].Form.FormTrigChrgRlyFailed := TRUE; 
			Trips_DB.Section[4].Form.FormTrigChrgRlyFaultDelay_TON (IN:= FALSE);
		END_IF;
	ELSE
		Trips_DB.Section[4].Form.FormTrigChrgRlyFaultDelay_TON (IN:= FALSE);
END_IF;

//preform trigger charge
		//fail to close
IF (LCP.Section[4].Form.ClosePreFormTrigChargeRly = TRUE AND LCP.Section[4].Form.PreFormTrigChargeRly_close = FALSE) OR 
		(LCP.Section[4].Form.ClosePreFormTrigChargeRly = FALSE AND LCP.Section[4].Form.PreFormTrigChargeRly_close = TRUE) 
		THEN 
		//start timer
		Trips_DB.Section[4].Form.PreFormTrigChrgRlyFaultDelay_TON (IN:= TRUE, PT := ChrgRlyFaultDelay_PT);
		
		IF Trips_DB.Section[4].Form.PreFormTrigChrgRlyFaultDelay_TON.Q = TRUE THEN 
			Trips_DB.Section[4].Form.PreFormTrigChrgRlyFailed := TRUE; 
			Trips_DB.Section[4].Form.PreFormTrigChrgRlyFaultDelay_TON (IN:= FALSE);
		END_IF;
	ELSE
		Trips_DB.Section[4].Form.PreFormTrigChrgRlyFaultDelay_TON (IN:= FALSE);
END_IF;

//preform dump
	//fail to close
IF (LCP.Section[4].Form.OpenPreFormDumpRly = TRUE AND LCP.Section[4].Form.PreFormDumpRly_close = FALSE) OR 
		(LCP.Section[4].Form.OpenPreFormDumpRly = FALSE AND LCP.Section[4].Form.PreFormDumpRly_close = TRUE) 
		THEN 
		//start timer
		Trips_DB.Section[4].Form.PreFormDumpRlyFaultDelay_TON (IN:= TRUE, PT := DumpRlyFaultDelay_PT);
		
		IF Trips_DB.Section[4].Form.PreFormDumpRlyFaultDelay_TON.Q = TRUE THEN 
			Trips_DB.Section[4].Form.PreFormDumpRlyFailed := TRUE; 
			Trips_DB.Section[4].Form.PreFormDumpRlyFaultDelay_TON (IN:= FALSE);
		END_IF;
	ELSE
		Trips_DB.Section[4].Form.PreFormDumpRlyFaultDelay_TON (IN:= FALSE);
END_IF;

//form trigger dump
	//fail to close
IF (LCP.Section[4].Form.OpenFormTrigDumpRly1 = TRUE AND LCP.Section[4].Form.FormTrigDumpRly1_close = FALSE) OR 
		(LCP.Section[4].Form.OpenFormTrigDumpRly1 = FALSE AND LCP.Section[4].Form.FormTrigDumpRly1_close = TRUE) 
		THEN 
		//start timer
		Trips_DB.Section[4].Form.FormTrigDumpRlyFaultDelay_TON (IN:= TRUE, PT := DumpRlyFaultDelay_PT);
		
		IF Trips_DB.Section[4].Form.FormTrigDumpRlyFaultDelay_TON.Q = TRUE THEN 
			Trips_DB.Section[4].Form.FormTrigDumpRly1Failed := TRUE; 
			Trips_DB.Section[4].Form.FormTrigDumpRlyFaultDelay_TON (IN:= FALSE);
		END_IF;
	ELSE
		Trips_DB.Section[4].Form.FormTrigDumpRlyFaultDelay_TON (IN:= FALSE);
END_IF;
	
//preform trigger dump
	//fail to close
IF (LCP.Section[4].Form.OpenPreFormTrigDumpRly1 = TRUE AND LCP.Section[4].Form.PreFormTrigDumpRly1_close = FALSE) OR 
		(LCP.Section[4].Form.OpenPreFormTrigDumpRly1 = FALSE AND LCP.Section[4].Form.PreFormTrigDumpRly1_close = TRUE) 
		THEN 
		//start timer
		Trips_DB.Section[4].Form.PreFormTrigDumpRlyFaultDelay_TON (IN:= TRUE, PT := DumpRlyFaultDelay_PT);
		
		IF Trips_DB.Section[4].Form.PreFormTrigDumpRlyFaultDelay_TON.Q = TRUE THEN 
			Trips_DB.Section[4].Form.PreFormTrigDumpRly1Failed := TRUE; 
			Trips_DB.Section[4].Form.PreFormTrigDumpRlyFaultDelay_TON (IN:= FALSE);
		END_IF;
	ELSE
		Trips_DB.Section[4].Form.PreFormTrigDumpRlyFaultDelay_TON (IN:= FALSE);
END_IF;
	

// if rly fail to close or fail to open then trips_db.rly_failed - for alarms	
FOR j := 1 TO 3 BY 1 DO
	//peak
	IF Trips_DB.Section[j].Peak.ChargeRelay1_FailtoClose = TRUE OR Trips_DB.Section[j].Peak.ChargeRelay1_FailtoOpen = TRUE THEN
		Trips_DB.Section[j].Peak.ChargeRelay1_Failed := TRUE;  
	END_IF;
	
	IF Trips_DB.Section[j].Peak.ChargeRelay2_FailtoClose = TRUE OR Trips_DB.Section[j].Peak.ChargeRelay2_FailtoOpen = TRUE THEN
		Trips_DB.Section[j].Peak.ChargeRelay2_Failed := TRUE;  
	END_IF;
	
	IF Trips_DB.Section[j].Peak.DumpRelay1_FailtoClose = TRUE OR Trips_DB.Section[j].Peak.DumpRelay1_FailtoOpen = TRUE THEN
		Trips_DB.Section[j].Peak.DumpRelay1_Failed := TRUE;  
	END_IF;
	
	IF Trips_DB.Section[j].Peak.DumpRelay2_FailtoClose = TRUE OR Trips_DB.Section[j].Peak.DumpRelay2_FailtoOpen = TRUE THEN
		Trips_DB.Section[j].Peak.DumpRelay2_Failed := TRUE;  
	END_IF;
	
	//sust
	IF Trips_DB.Section[j].Sust.ChargeRelay1_FailtoClose = TRUE OR Trips_DB.Section[j].Sust.ChargeRelay1_FailtoOpen = TRUE THEN
		Trips_DB.Section[j].Sust.ChargeRelay1_Failed := TRUE;  
	END_IF;
	
	IF Trips_DB.Section[j].Sust.ChargeRelay2_FailtoClose = TRUE OR Trips_DB.Section[j].Sust.ChargeRelay2_FailtoOpen = TRUE THEN
		Trips_DB.Section[j].Sust.ChargeRelay2_Failed := TRUE;  
	END_IF;
	
	IF Trips_DB.Section[j].Sust.DumpRelay1_FailtoClose = TRUE OR Trips_DB.Section[j].Sust.DumpRelay1_FailtoOpen = TRUE THEN
		Trips_DB.Section[j].Sust.DumpRelay1_Failed := TRUE;  
	END_IF;
	
	IF Trips_DB.Section[j].Sust.DumpRelay2_FailtoClose = TRUE OR Trips_DB.Section[j].Sust.DumpRelay2_FailtoOpen = TRUE THEN
		Trips_DB.Section[j].Sust.DumpRelay2_Failed := TRUE;  
	END_IF;
	
END_FOR;

//any system tripped
FOR k := 1 TO 4 BY 1 DO
	IF Trips_DB.Section[k].SystemTripped = TRUE OR Trips_DB.MCPsystemTripped = TRUE THEN
		Trips_DB.AnySystemTripped := TRUE;
		ELSE
			Trips_DB.AnySystemTripped := FALSE;
	END_IF;
END_FOR

// no faulted detected
IF (Trips_DB.AnySystemTripped = FALSE AND
	Trips_DB.AnyChargerOverTemp = FALSE AND
	Trips_DB.AnyChargerLoadFault = FALSE AND  //no charger fault is a permissives to charge
	Trips_DB.AnyChargerInterlockOpen = FALSE AND
	Trips_DB.AnyChargerFaulted = FALSE AND
	Trips_DB.AnyEstopPressed = FALSE AND
	Trips_DB.AnyDumpRlyFail = FALSE AND
	Trips_DB.AnyChargeRlyFail = FALSE AND 
	Trips_DB.AllDCpsuOK = TRUE AND
	Trips_DB.AnyLossInhibitSignal = FALSE AND
	Trips_DB.AnyLossHVONsignal = FALSE AND 
	Trips_DB.MachineGNDrlyFailed = FALSE AND 
	Trips_DB.ChargingTimerRunout = FALSE AND
	Trips_DB.ChargedTimerRunout = FALSE AND
	Trips_DB.DumpTimerRunout) OR HMI_DB.NoFaultDetectedBP = TRUE //admin bypass
	THEN
		Trips_DB.NoFaultDetected := TRUE;
	ELSE
		Trips_DB.NoFaultDetected := FALSE;
END_IF;


(*
FOR i := 1 TO 10 BY 1 DO
	IF (Trips_DB.Coil[i].ACInterlockRelayFailedtoClose = TRUE OR 
		Trips_DB.Coil[i].ACInterlockRelayFailedtoOpen = TRUE OR 
		Trips_DB.Coil[i].ChargeRelay_FailtoClose = TRUE OR
		Trips_DB.Coil[i].ChargeRelay_FailtoOpen = TRUE OR
		Trips_DB.Coil[i].DumpRelay1_FailtoClose =  TRUE OR 
		Trips_DB.Coil[i].DumpRelay1_FailtoOpen = TRUE OR 
		Trips_DB.Coil[i].DumpRelay2_FailtoClose =  TRUE OR 
		Trips_DB.Coil[i].DumpRelay2_FailtoOpen = TRUE OR 
		Trips_DB.Coil[i].ChargerVoltageReadingFaulted = TRUE OR
		Trips_DB.Coil[i].CurrentReadingFaulted = TRUE OR
		Devices.Coil[i].Local_EstopPB_Pressed = TRUE OR
		Devices.Coil[i].LossPneumaticPressure = FALSE) AND Devices.Coil[i].CoilEnabled = TRUE 	
		THEN
			Devices.Coil[i].SystemFaulted := TRUE;
	END_IF
	
	IF Devices.Coil[i].SystemFaulted = TRUE THEN
		Trips_DB.SystemTripped := TRUE;
	END_IF;
END_FOR;

//*********************************** Test
(*IF InstrumentReading.R2_01_CH01 <= 0.0 THEN
	delay2s(input := FALSE);
ELSE 
	delay2s (input := TRUE);
END_IF;
bTest := delay2s.output;
*)
// Instrumentation Hardware trip
//Input.R2_01_00_Status.0;
*)
//************** Clear System Fault
IF Trips_DB.ClearAllFaults = TRUE OR stControl.ClearAllFaults = TRUE THEN
	//Trips_DB.InstrumentationFaulted := FALSE;

	Trips_DB.MCPsystemTripped := FALSE; //reset mcp trip
	Trips_DB.AnyChargerOverTemp := FALSE;
	Trips_DB.AnyChargerLoadFault := FALSE;  
	Trips_DB.AnyChargerInterlockOpen := FALSE;
	Trips_DB.AnyChargerFaulted := FALSE;
	Trips_DB.AnyEstopPressed := FALSE;
	Trips_DB.AnyDumpRlyFail := FALSE;
	Trips_DB.AnyChargeRlyFail := FALSE;
	Trips_DB.MasterStopPBPressed := FALSE; //this is only for alarms
	Trips_DB.CageEStopCircuitBroken := FALSE;
	Trips_DB.MCPLossDCpower := FALSE;
	Trips_DB.AnyLossInhibitSignal := FALSE;
	Trips_DB.AnyLossHVONsignal := FALSE;
	Trips_DB.MachineGNDrlyFailed := FALSE;
	Trips_DB.ChargingTimerRunout := FALSE;
	Trips_DB.ChargedTimerRunout  := FALSE;
	Trips_DB.DumpTimerRunout := FALSE;
	//Trips_DB.AnyACInterlockFail := FALSE;
	//reset relay trips
	FOR j := 1 TO 3 BY 1 DO 
		//reset relay faults
		Trips_DB.Section[j].SystemTripped := FALSE;
		//Peaking
		Trips_DB.Section[j].Peak.DumpRelay1_FailtoClose := FALSE;
		Trips_DB.Section[j].Peak.DumpRelay1_FailtoOpen := FALSE;
		Trips_DB.Section[j].Peak.DumpRelay2_FailtoClose := FALSE;
		Trips_DB.Section[j].Peak.DumpRelay2_FailtoOpen := FALSE;
		Trips_DB.Section[j].Peak.ChargeRelay1_FailtoClose := FALSE;
		Trips_DB.Section[j].Peak.ChargeRelay1_FailtoOpen := FALSE;
		Trips_DB.Section[j].Peak.ChargeRelay2_FailtoClose := FALSE;
		Trips_DB.Section[j].Peak.ChargeRelay2_FailtoOpen := FALSE;
		//Sust
		Trips_DB.Section[j].Sust.DumpRelay1_FailtoClose := FALSE;
		Trips_DB.Section[j].Sust.DumpRelay1_FailtoOpen := FALSE;
		Trips_DB.Section[j].Sust.DumpRelay2_FailtoClose := FALSE;
		Trips_DB.Section[j].Sust.DumpRelay2_FailtoOpen := FALSE;
		Trips_DB.Section[j].Sust.ChargeRelay1_FailtoClose := FALSE;
		Trips_DB.Section[j].Sust.ChargeRelay1_FailtoOpen := FALSE;
		Trips_DB.Section[j].Sust.ChargeRelay2_FailtoClose := FALSE;
		Trips_DB.Section[j].Sust.ChargeRelay2_FailtoOpen := FALSE;
	
	END_FOR;
	
	//FORM
	Trips_DB.Section[4].Form.ChargeRelay1_FailtoOpen := FALSE;
	Trips_DB.Section[4].Form.ChargeRelay1_FailtoClose := FALSE;
	Trips_DB.Section[4].Form.ChargeRelay1_Failed:= FALSE;
	Trips_DB.Section[4].Form.ChargeRelay2_FailtoOpen := FALSE;
	Trips_DB.Section[4].Form.ChargeRelay2_FailtoClose := FALSE;
	Trips_DB.Section[4].Form.ChargeRelay2_Failed:= FALSE;
	
	Trips_DB.Section[4].Form.DumpRelay1_FailtoOpen := FALSE;
	Trips_DB.Section[4].Form.DumpRelay1_FailtoClose := FALSE;
	Trips_DB.Section[4].Form.DumpRelay1_Failed := FALSE;
	Trips_DB.Section[4].Form.DumpRelay2_FailtoOpen := FALSE;
	Trips_DB.Section[4].Form.DumpRelay2_FailtoClose := FALSE;
	Trips_DB.Section[4].Form.DumpRelay2_Failed := FALSE;
	
	Trips_DB.Section[4].Form.PreFormChrgRlyFailed := FALSE;
	Trips_DB.Section[4].Form.FormTrigChrgRlyFailed := FALSE;
	Trips_DB.Section[4].Form.PreFormTrigChrgRlyFailed := FALSE;
	Trips_DB.Section[4].Form.PreFormDumpRlyFailed := FALSE;
	Trips_DB.Section[4].Form.FormTrigDumpRly1Failed := FALSE;
	Trips_DB.Section[4].Form.PreFormTrigDumpRly1Failed := FALSE;
	
	Trips_DB.Section[4].SystemTripped := FALSE;
	
	evtLogger.ClearAllAlarms(0, FALSE);
	//evtLogger.ClearLoggedEvents(1);
END_IF;


//IF i > 8 THEN 
IF i > 3 THEN
	i := 1;
END_IF;

IF j > 3 THEN 
	j := 1;
END_IF;

IF k > 4 THEN 
	k := 1;
END_IF;

END_PROGRAM

// ---- POUs/Sequence.TcPOU
PROGRAM Sequence
VAR
	ePulseState : E_PulseState;
	eCommand	: E_Command;
	eStatus		: E_Status;
	
	ChargeRlyDelayON_Timer  : TON;
	ChargeRlyDelayDONE		: BOOL;
	ChargeRlyDelayON_PT		: TIME := T#250MS; //used for delay close and delay open for safe mode
	AbortPSnRlyDelay_Timer	: TON;
	AbortPSnRlyDelay_PT		: TIME := T#5MS; //defualt is 5ms
	AbortPSnRlyDelayDONE	: BOOL;
	ChargeCompleted			: BOOL;
	ChargingRunOutTMR_TON	: TON;
	ChargingRunOutTMR_ET	: TIME;
	ChargedRunOutTMR_TON	: TON;
	ChargedRunOutTMR_ET		: TIME;
	
	DumpingRunOutTMR_TON 	: TON;
	DumpingRunOutTMR_PT		: TIME := T#180S;
	DumpingRunOutTMR_ET		: TIME;
	LocalDumpActive			: BOOL := FALSE;
	Dump					: Dump_FB;	
	LocalDumpElapse			: REAL;				
		
	ReadyToCharge 			: BOOL;
	StartChargingBroadcast	: BOOL := FALSE;
	StartCharger			: ARRAY[1..8] OF BOOL;
	StartGLS3Charger		: BOOL;
	
	SparkGapCharger_TON		: TON;
	SparkGapCharger_PT		: TIME := T#1S;
	SparkGapCharger_ET		: TIME;
	
	i : INT := 1; // charger 1-8
	j : INT := 1; // section 1 - 3
	k : INT := 1;
	
	ChargeTimeFinished		: BOOL;
END_VAR

//Critical Delay Time
HMI_DB.ChargerHVOFF_rlyDelayPT := INT_TO_TIME(HMI_DB.ChargerHVOFF_rlyDelayPT_INT);
AbortPSnRlyDelay_PT := HMI_DB.ChargerHVOFF_rlyDelayPT;

//hv output delay
HMI_DB.HVONdelayPT := INT_TO_TIME (HMI_DB.HVONdelayPT_INT);
ChargeRlyDelayON_PT := HMI_DB.HVONdelayPT;

//runout timer
HMI_DB.RunOutTMR_PT := INT_TO_TIME (HMI_DB.RunOutTMR_PT_INT*1000);
HMI_DB.RunOutTMR_elapse := (TIME_TO_INT (HMI_DB.RunOutTMR_PT - ChargedRunOutTMR_TON.ET))/1000;
HMI_DB.ChargingRunOutTMR_elapse := TIME_TO_INT(ChargingRunOutTMR_TON.PT/1000 - ChargingRunOutTMR_TON.ET/1000);

//charge realy timer 
ChargeRlyDelayON_Timer(PT := ChargeRlyDelayON_PT);

//screen room asks to go to idle, it will go to safe state. 
//GVL.RemoteModeSelected is MCP_IO.RemoteModeSelected OR HMI_DB.RemoteModeSelected 
IF GVL.RemoteModeSelected = TRUE AND eCommand = E_Command.IDLE AND Trips_DB.NoFaultDetected = TRUE 
	THEN
		ePulseState := E_PulseState.SAFE;
END_IF;
	//at anypoint if screen room wants abort or hmi abort pb is pressed
IF eCommand = E_Command.ABORT OR HMI_DB.AbortPB = TRUE //OR Trips_DB.AnyEstopPressed = TRUE 
	THEN
	 	ePulseState := E_PulseState.ABORT;
END_IF;

IF Trips_DB.NoFaultDetected = FALSE 
	THEN
		ePulseState := E_PulseState.TRIPPED;
END_IF;

IF GVL.RemoteModeSelected = FALSE AND Trips_DB.NoFaultDetected = TRUE 
	THEN
		ePulseState := E_PulseState.LOCALMODE;
END_IF;

//lift machine GND
IF Permissives_DB.AllSectCapsDischarged = FALSE THEN //at least one cap has voltage >10V
	MCP_IO.LiftMachineGND := TRUE;
	ELSE
		MCP_IO.LiftMachineGND := FALSE;
END_IF;

//reset timer
IF ePulseState <> E_PulseState.CHARGING THEN 
	ChargingRunOutTMR_TON (IN := FALSE);
	//FOR i := 1 TO 8 BY 1 DO 
	FOR i := 1 TO 3 BY 1 DO
		ChargeTime_DB.ChargerDelay_TON[i] (IN := FALSE, PT := ChargeTime_DB.ChargerDelay_PT[i], ET => ChargeTime_DB.ChargerDelay_ET[i]);
		ChargeTime_DB.ChargingTimeElapse_TON[i].IN := FALSE;
		ChargeRlyDelayON_Timer (IN := FALSE);
	END_FOR;
	ChargeTime_DB.PreFormChargeTime_TON (IN := FALSE, PT := ChargeTime_DB.PreFormChargeTime_PT, ET => ChargeTime_DB.PreFormChargeTime_ET);
	ChargeTime_DB.PreFormChargingTimeElapse_TON.IN := FALSE;
END_IF
IF ePulseState <> (E_PulseState.CHARGECOMPLETE OR E_PulseState.DISCONNECTING) THEN 
	ChargedRunOutTMR_TON (IN := FALSE); // only needed in charge complete
END_IF

CASE ePulseState OF 
	
	//Safe OR IDLE
	E_PulseState.SAFE: 
					//TURN OFF ALL CHARGERS
					//FOR i := 1 TO 8 BY 1 DO 
					FOR i := 1 TO 3 BY 1 DO 
						MCP_IO.Charger[i].inhibit := TRUE; // inhibit = high, no output | inhibit = low, allows output
						MCP_IO.Charger[i].HV_ON := FALSE; 
						MCP_IO.Charger[i].voltageSP := 0;
						StartCharger[i] := FALSE; // reset bit
						ChargeTimeFinished := FALSE;
						StartChargingBroadcast := FALSE;
						//reset charger delay timer
						ChargeTime_DB.ChargerDelay_TON[i] (IN := FALSE, PT := ChargeTime_DB.ChargerDelay_PT[i], ET => ChargeTime_DB.ChargerDelay_ET[i]);
						ChargeTime_DB.ChargingTimeElapse_TON[i] (IN := FALSE); 
					END_FOR;
					StartGLS3Charger := FALSE;
					ChargeTime_DB.PreFormChargeTime_TON (IN := FALSE, PT := ChargeTime_DB.PreFormChargeTime_PT, ET => ChargeTime_DB.PreFormChargeTime_ET);
					MCP_IO.GLS1_hvON := FALSE;
					MCP_IO.GLS2_hvON := FALSE;
					MCP_IO.GLS3_hvON := FALSE;
					MCP_IO.GLS1_voltageSP := 0;
					MCP_IO.GLS2_voltageSP := 0;
					MCP_IO.GLS3_voltageSP := 0;
					SparkGapCharger_TON(IN := FALSE);
					//start delay
					IF Permissives_DB.AllChargerHVisON = FALSE THEN 
						ChargeRlyDelayON_Timer (IN := TRUE, PT := ChargeRlyDelayON_PT);	
						ELSE
							ChargeRlyDelayON_Timer (IN := FALSE, PT := ChargeRlyDelayON_PT);				
					END_IF;
					
					IF ChargeRlyDelayON_Timer.Q = TRUE THEN 
						ChargeRlyDelayDONE := TRUE;
						ChargeRlyDelayON_Timer (IN := FALSE);
					END_IF;
					IF ChargeRlyDelayDONE = TRUE THEN
						FOR j := 1 TO 3 BY 1 DO 
							//Open all charge relays after 250ms
							LCP.Section[j].Peak.CloseChargeRelay1 := FALSE; 
							LCP.Section[j].Peak.CloseChargeRelay2 := FALSE; 
							LCP.Section[j].Sust.CloseChargeRelay1 := FALSE;
							LCP.Section[j].Sust.CloseChargeRelay2 := FALSE;
							//close all dump relays  - for SAFE STATE they can all go together
							LCP.Section[j].Peak.OpenDumpRelay1 := FALSE;
							LCP.Section[j].Peak.OpenDumpRelay2 := FALSE;
							LCP.Section[j].Sust.OpenDumpRelay1 := FALSE;
							LCP.Section[j].Sust.OpenDumpRelay2 := FALSE;	
						END_FOR;
						//open all charge rly on form
						LCP.Section[4].Form.CloseChargeRelay1 := FALSE;
						LCP.Section[4].Form.CloseChargeRelay2 := FALSE;
						LCP.Section[4].Form.CloseFormTrigChargeRly := FALSE;
						LCP.Section[4].Form.ClosePreFormChargeRly := FALSE;
						LCP.Section[4].Form.ClosePreFormTrigChargeRly := FALSE;
						//close all dump relay on form
						LCP.Section[4].Form.OpenDumpRelay1 := FALSE;
						LCP.Section[4].Form.OpenDumpRelay2 := FALSE;
						LCP.Section[4].Form.OpenPreFormDumpRly := FALSE;
						LCP.Section[4].Form.OpenFormTrigDumpRly1 := FALSE;
						LCP.Section[4].Form.OpenPreFormTrigDumpRly1 := FALSE;
						
						ChargeRlyDelayDONE := FALSE;
						ChargeRlyDelayON_Timer (IN := FALSE);
					END_IF;
					// short contacts engaged as a permissives to say it is safe???????
					//send status to screen room
					eStatus := E_Status.SAFE;
					
					IF Trips_DB.NoFaultDetected = TRUE AND 
						Permissives_DB.NoShortingUnknowns AND 
						Permissives_DB.AllShortContactEngaged = FALSE
						THEN 
							ReadyToCharge := TRUE;
							ELSE
								ReadyToCharge := FALSE;		
					END_IF;
					//wait for command from screen room
					IF GVL.RemoteModeSelected = TRUE AND ReadyToCharge = TRUE AND eCommand = E_Command.CHARGE 
						THEN
							ePulseState := E_PulseState.CHARGING;
						//ELSIF MCP_IO.RemoteModeSelected = TRUE AND eCommand = E_Command.IDLE THEN
							//ePulseState := E_PulseState.SAFE;
						ELSIF MCP_IO.RemoteModeSelected = TRUE AND eCommand = E_Command.DUMP THEN
							ePulseState := E_PulseState.DUMPING;
					END_IF;
					ChargingRunOutTMR_TON (IN := FALSE);
					ChargedRunOutTMR_TON (IN := FALSE);
					DumpingRunOutTMR_TON (IN := FALSE);
	//Charging
	E_PulseState.CHARGING: 
					MCP_IO.LiftMachineGND := TRUE; //call the bit again in case it did not lift
					
					IF Recipe.PeakSupplyEN = FALSE THEN
						MCP_IO.Charger[1].voltageSP := 0;
						MCP_IO.Charger[2].voltageSP := 0;
						MCP_IO.Charger[3].voltageSP := 0;
					END_IF
					(*IF Recipe.SustSupplyEN = FALSE THEN
						MCP_IO.Charger[4].voltageSP := 0;
						MCP_IO.Charger[5].voltageSP := 0;
						MCP_IO.Charger[6].voltageSP := 0;
					END_IF
					IF Recipe.FormSupplyEN = FALSE THEN
						MCP_IO.Charger[7].voltageSP := 0;
						MCP_IO.Charger[8].voltageSP := 0;
					END_IF*)
					IF Recipe.PFormSupplyEN = FALSE THEN
						MCP_IO.GLS3_voltageSP := 0;
					END_IF
					
					//start charging runout timer
					ChargingRunOutTMR_TON (IN := TRUE, PT := (ChargeTime_DB.LongestChargeTime_PT + HMI_DB.RunOutTMR_PT), ET => ChargingRunOutTMR_ET);
	
					//will need the charge time sequence to see stagger each bank's charge time......done
					IF Trips_DB.NoFaultDetected = TRUE THEN 
						FOR j := 1 TO 3 BY 1 DO 
							//Open all dump relays  
							LCP.Section[j].Peak.OpenDumpRelay1 := TRUE;
							LCP.Section[j].Peak.OpenDumpRelay2 := TRUE;
							LCP.Section[j].Sust.OpenDumpRelay1 := TRUE;
							LCP.Section[j].Sust.OpenDumpRelay2 := TRUE;	
						END_FOR;
						//open all dump relay on form
						LCP.Section[4].Form.OpenDumpRelay1 := TRUE;
						LCP.Section[4].Form.OpenDumpRelay2 := TRUE;
						LCP.Section[4].Form.OpenPreFormDumpRly := TRUE;
						LCP.Section[4].Form.OpenFormTrigDumpRly1 := TRUE;
						LCP.Section[4].Form.OpenPreFormTrigDumpRly1 := TRUE;
						//if all dump relays open then close charger relays
						IF Permissives_DB.AllDumpRelaysOpen = TRUE THEN 
							//close all charge rly 
							FOR j := 1 TO 3 BY 1 DO
								IF Recipe.PeakSupplyEN THEN
									LCP.Section[j].Peak.CloseChargeRelay1 := TRUE; 
									LCP.Section[j].Peak.CloseChargeRelay2 := TRUE; 
									ELSE
										LCP.Section[j].Peak.CloseChargeRelay1 := FALSE; 
										LCP.Section[j].Peak.CloseChargeRelay2 := FALSE; 
								END_IF;
								IF Recipe.SustSupplyEN THEN
									LCP.Section[j].Sust.CloseChargeRelay1 := TRUE;
									LCP.Section[j].Sust.CloseChargeRelay2 := TRUE;
									ELSE
										LCP.Section[j].Sust.CloseChargeRelay1 := FALSE;
										LCP.Section[j].Sust.CloseChargeRelay2 := FALSE;
								END_IF
							END_FOR;
							//close all charge rly on form
							IF Recipe.FormSupplyEN THEN
								LCP.Section[4].Form.CloseChargeRelay1 := TRUE;
								LCP.Section[4].Form.CloseChargeRelay2 := TRUE;
								LCP.Section[4].Form.CloseFormTrigChargeRly := TRUE;
								ELSE
									LCP.Section[4].Form.CloseChargeRelay1 := FALSE;
									LCP.Section[4].Form.CloseChargeRelay2 := FALSE;
									LCP.Section[4].Form.CloseFormTrigChargeRly := FALSE;
							END_IF
							
							IF Recipe.PFormSupplyEN THEN
								LCP.Section[4].Form.ClosePreFormChargeRly := TRUE;
								LCP.Section[4].Form.ClosePreFormTrigChargeRly := TRUE;
								ELSE
									LCP.Section[4].Form.ClosePreFormChargeRly := FALSE;
									LCP.Section[4].Form.ClosePreFormTrigChargeRly := FALSE;
							END_IF
						END_IF;	
					END_IF;
					
					IF Trips_DB.NoFaultDetected = TRUE AND Permissives_DB.AllChargeRelaysClosed = TRUE 
						THEN 
							ChargeRlyDelayON_Timer (IN := TRUE, PT := ChargeRlyDelayON_PT);
							ELSE
								ChargeRlyDelayON_Timer (IN := FALSE, PT := ChargeRlyDelayON_PT);
					END_IF;
					//start broadcasting on charger timer
					IF ChargeRlyDelayON_Timer.Q = TRUE THEN 
						StartChargingBroadcast := TRUE;
					END_IF;
					//start timer 
					IF StartChargingBroadcast = TRUE THEN 
						//start total charge time TIMER
						ChargeTime_DB.LongestChargeTime_TON (IN := TRUE, PT := ChargeTime_DB.LongestChargeTime_PT, ET => ChargeTime_DB.LongestChargeTime_ET);
						//Turn inhibit On on all chargers and start timer
						(*FOR i := 1 TO 8 BY 1 DO 
							//MCP_IO.Charger[i].inhibit := TRUE; 
							// delay stagger starts here 
							//ChargeTime_DB.ChargerDelay_TON[i] (IN := TRUE, PT := ChargeTime_DB.ChargerDelay_PT[i], ET => ChargeTime_DB.ChargerDelay_ET[i]);
						END_FOR;*)
						//send voltage SP to chargers
						IF Recipe.PeakSupplyEN = TRUE THEN
							MCP_IO.Charger[1].voltageSP := REAL_TO_DINT (Setpoints.TDKLoad[1].RequiredChargedV * 1000);
							MCP_IO.Charger[2].voltageSP := REAL_TO_DINT (Setpoints.TDKLoad[2].RequiredChargedV * 1000);
							MCP_IO.Charger[3].voltageSP := REAL_TO_DINT (Setpoints.TDKLoad[3].RequiredChargedV * 1000);
							END_IF;
						(*IF Recipe.SustSupplyEN = TRUE THEN
							MCP_IO.Charger[4].voltageSP := REAL_TO_DINT (Setpoints.TDKLoad[4].RequiredChargedV * 1000);
							MCP_IO.Charger[5].voltageSP := REAL_TO_DINT (Setpoints.TDKLoad[5].RequiredChargedV * 1000);
							MCP_IO.Charger[6].voltageSP := REAL_TO_DINT (Setpoints.TDKLoad[6].RequiredChargedV * 1000);
							END_IF;
						IF Recipe.FormSupplyEN = TRUE THEN
							MCP_IO.Charger[7].voltageSP := REAL_TO_DINT (Setpoints.TDKLoad[7].RequiredChargedV * 1000);
							MCP_IO.Charger[8].voltageSP := REAL_TO_DINT (Setpoints.TDKLoad[8].RequiredChargedV * 1000);
							END_IF;*)
						IF Recipe.PFormSupplyEN = TRUE THEN
							MCP_IO.GLS3_voltageSP := REAL_TO_DINT (Setpoints.GLSLoad.RequiredChargedV * 1000);
							END_IF
						MCP_IO.GLS1_voltageSP := REAL_TO_DINT (Setpoints.GLS1_VSP * 1000);
						MCP_IO.GLS2_voltageSP := REAL_TO_DINT (Setpoints.GLS2_VSP * 1000);
						
						// delay stagger starts here 
						IF Recipe.PeakSupplyEN = TRUE THEN
							ChargeTime_DB.ChargerDelay_TON[1] (IN := TRUE, PT := ChargeTime_DB.ChargerDelay_PT[1], ET => ChargeTime_DB.ChargerDelay_ET[1]);
							ChargeTime_DB.ChargerDelay_TON[2] (IN := TRUE, PT := ChargeTime_DB.ChargerDelay_PT[2], ET => ChargeTime_DB.ChargerDelay_ET[2]);
							ChargeTime_DB.ChargerDelay_TON[3] (IN := TRUE, PT := ChargeTime_DB.ChargerDelay_PT[3], ET => ChargeTime_DB.ChargerDelay_ET[3]);
						END_IF
						(*IF Recipe.SustSupplyEN = TRUE THEN
							ChargeTime_DB.ChargerDelay_TON[4] (IN := TRUE, PT := ChargeTime_DB.ChargerDelay_PT[4], ET => ChargeTime_DB.ChargerDelay_ET[4]);
							ChargeTime_DB.ChargerDelay_TON[5] (IN := TRUE, PT := ChargeTime_DB.ChargerDelay_PT[5], ET => ChargeTime_DB.ChargerDelay_ET[5]);
							ChargeTime_DB.ChargerDelay_TON[6] (IN := TRUE, PT := ChargeTime_DB.ChargerDelay_PT[6], ET => ChargeTime_DB.ChargerDelay_ET[6]);
						END_IF
						IF Recipe.FormSupplyEN = TRUE THEN
							ChargeTime_DB.ChargerDelay_TON[7] (IN := TRUE, PT := ChargeTime_DB.ChargerDelay_PT[7], ET => ChargeTime_DB.ChargerDelay_ET[7]);
							ChargeTime_DB.ChargerDelay_TON[8] (IN := TRUE, PT := ChargeTime_DB.ChargerDelay_PT[8], ET => ChargeTime_DB.ChargerDelay_ET[8]);							
						END_IF*)
						IF Recipe.PFormSupplyEN = TRUE THEN
							ChargeTime_DB.PreFormChargeTime_TON (IN := TRUE, PT := ChargeTime_DB.PreFormChargeTime_PT, ET => ChargeTime_DB.PreFormChargeTime_ET);
						END_IF						
						ChargeRlyDelayON_Timer (IN := FALSE);
						SparkGapCharger_TON(IN := TRUE, PT := (ChargeTime_DB.LongestChargeTime_PT-SparkGapCharger_PT), ET => SparkGapCharger_ET);
					ELSE
						//Turn inhibit High on all chargers and turn off all timer if no broadcasting
						//FOR i := 1 TO 8 BY 1 DO 
						FOR i := 1 TO 3 BY 1 DO
							MCP_IO.Charger[i].inhibit := TRUE; 
							// turn off timer
							ChargeTime_DB.ChargerDelay_TON[i] (IN := FALSE, PT := ChargeTime_DB.ChargerDelay_PT[i], ET => ChargeTime_DB.ChargerDelay_ET[i]);
						END_FOR;
						ChargeTime_DB.PreFormChargeTime_TON (IN := FALSE, PT := ChargeTime_DB.PreFormChargeTime_PT, ET => ChargeTime_DB.PreFormChargeTime_ET);	
						ChargeTime_DB.LongestChargeTime_TON (IN := FALSE); //reset timer	
						SparkGapCharger_TON(IN := TRUE);						
					END_IF;
					
					//turn on HV output to load	
					IF Recipe.PeakSupplyEN = TRUE AND ChargeTime_DB.ChargerDelay_TON[1].Q = TRUE THEN
						StartCharger[1] := TRUE;
					END_IF
					IF Recipe.PeakSupplyEN = TRUE AND ChargeTime_DB.ChargerDelay_TON[2].Q = TRUE THEN
						StartCharger[2] := TRUE;
					END_IF
					IF Recipe.PeakSupplyEN = TRUE AND ChargeTime_DB.ChargerDelay_TON[3].Q = TRUE THEN
						StartCharger[3] := TRUE;
					END_IF
					(*IF Recipe.SustSupplyEN = TRUE AND ChargeTime_DB.ChargerDelay_TON[4].Q = TRUE THEN
						StartCharger[4] := TRUE;
					END_IF
					IF Recipe.SustSupplyEN = TRUE AND ChargeTime_DB.ChargerDelay_TON[5].Q = TRUE THEN
						StartCharger[5] := TRUE;
					END_IF
					IF Recipe.SustSupplyEN = TRUE AND ChargeTime_DB.ChargerDelay_TON[6].Q = TRUE THEN
						StartCharger[6] := TRUE;
					END_IF
					IF Recipe.FormSupplyEN = TRUE AND ChargeTime_DB.ChargerDelay_TON[7].Q = TRUE THEN
						StartCharger[7] := TRUE;
					END_IF
					IF Recipe.FormSupplyEN = TRUE AND ChargeTime_DB.ChargerDelay_TON[8].Q = TRUE THEN
						StartCharger[8] := TRUE;
					END_IF*)

					
					//FOR k := 1 TO 8 BY 1 DO
					FOR k := 1 TO 3 BY 1 DO
						(*IF ChargeTime_DB.ChargerDelay_TON[k].Q = TRUE THEN
							StartCharger[k] := TRUE;
						END_IF;
						*)
						IF StartCharger[k] = TRUE THEN
							MCP_IO.Charger[k].HV_ON := TRUE; 
							MCP_IO.Charger[k].inhibit := FALSE;
							ChargeTime_DB.ChargerDelay_TON[k] (IN := FALSE, PT := ChargeTime_DB.ChargerDelay_PT[k], ET => ChargeTime_DB.ChargerDelay_ET[k]);
							//start time elapse
							ChargeTime_DB.ChargingTimeElapse_TON[k] (IN := TRUE, PT := REAL_TO_TIME (1000*MCP_IO.Charger[k].ChargeTime.timeToChargeLoad));
						END_IF;
						
						IF ChargeTime_DB.ChargingTimeElapse_TON[k].Q THEN
							StartCharger[k] := FALSE;
							ChargeTime_DB.ChargingTimeElapse_TON[k] (IN := FALSE); 
						END_IF;
					END_FOR
					//GLS 3
					IF ChargeTime_DB.PreFormChargeTime_TON.Q = TRUE AND Recipe.PFormSupplyEN = TRUE THEN
						StartGLS3Charger := TRUE;
					END_IF;
					IF StartGLS3Charger = TRUE THEN 
						MCP_IO.GLS3_hvON := TRUE;
						ChargeTime_DB.PreFormChargeTime_TON (IN := FALSE, PT := ChargeTime_DB.PreFormChargeTime_PT, ET => ChargeTime_DB.PreFormChargeTime_ET);
						//for hmi
						ChargeTime_DB.PreFormChargingTimeElapse_TON (IN := TRUE, PT :=  REAL_TO_TIME (1000*MCP_IO.GLS3_Load.timeToChargeLoad));
					END_IF;
					
					IF ChargeTime_DB.PreFormChargingTimeElapse_TON.Q = TRUE THEN
						StartGLS3Charger := FALSE;
						ChargeTime_DB.PreFormChargingTimeElapse_TON (IN := FALSE);
					END_IF
					
					IF SparkGapCharger_TON.Q = TRUE THEN 
						MCP_IO.GLS1_hvON := TRUE; //turn on spark gap charger
						MCP_IO.GLS2_hvON := TRUE;
						SparkGapCharger_TON(IN := FALSE);
					END_IF
					//turn off inhibit when HV is on
					(*IF Permissives_DB.AllChargerHVisON = TRUE THEN
						FOR i := 1 TO 8 BY 1 DO 
							MCP_IO.Charger[i].inhibit := FALSE; //start current output
						END_FOR;
						//StartChargingBroadcast := FALSE; // reset the broadcast bit whne all chargers 
					END_IF*)
					IF ChargingRunOutTMR_TON.Q = TRUE THEN
						Trips_DB.ChargingTimerRunout := TRUE;
						ChargingRunOutTMR_TON (IN := FALSE);
					END_IF
					
					IF Trips_DB.AnyLossHVONsignal = TRUE OR Trips_DB.ChargingTimerRunout = TRUE THEN 
						StartChargingBroadcast := FALSE; // reset the broadcast bit whne all chargers
						ChargeTimeFinished := FALSE; //reset chargetime done bit
						ChargingRunOutTMR_TON (IN := FALSE);
						//FOR i := 1 TO 8 BY 1 DO 
						FOR i := 1 TO 3 BY 1 DO 
							ChargeTime_DB.ChargingTimeElapse_TON[i] (IN := FALSE);							
						END_FOR
						ChargeTime_DB.PreFormChargingTimeElapse_TON (IN := FALSE);
						ePulseState := E_PulseState.TRIPPED; 
					END_IF
					//send status to screen room
					eStatus := E_Status.CHARGING;
					
					IF ChargeTime_DB.LongestChargeTime_TON.Q = TRUE THEN 
						ChargeTimeFinished := TRUE;
						ChargeTime_DB.LongestChargeTime_TON (IN := FALSE); //reset timer
					END_IF
					
					IF ChargeTimeFinished = TRUE THEN 
						//reset elapse timer
						//FOR i := 1 TO 8 BY 1 DO
						FOR i := 1 TO 3 BY 1 DO 
							StartCharger[i] := FALSE;
							ChargeTime_DB.ChargingTimeElapse_TON[i] (IN := FALSE);							
						END_FOR
						ChargeTime_DB.PreFormChargingTimeElapse_TON (IN := FALSE);
						StartGLS3Charger := FALSE;
						MCP_IO.GLS1_hvON := FALSE; //turn off spark gap charger
						MCP_IO.GLS2_hvON := FALSE;
						SparkGapCharger_TON(IN := FALSE);
					END_IF
					//condition for charge complete
					IF Permissives_DB.AllChargerEOC = TRUE AND ChargeTimeFinished = TRUE AND Permissives_DB.AllSectCapsFullyCharged = TRUE THEN 
						ChargeCompleted := TRUE;
						ELSE
							ChargeCompleted := FALSE;
					END_IF
					
					//if cap voltage feedback >= charger setpoints && EOC && all timer runout then chargecomplete
					IF ChargeCompleted = TRUE THEN 
						//FOR i := 1 TO 8 BY 1 DO
						FOR i := 1 TO 3 BY 1 DO 
							MCP_IO.Charger[i].HV_ON := FALSE; 
							MCP_IO.Charger[i].inhibit := TRUE;
							StartCharger[i] := FALSE;
							ChargeTime_DB.ChargingTimeElapse_TON[i] (IN := FALSE);	
							//ChargeTime_DB.ChargerDelay_TON[i] (IN := FALSE, PT := ChargeTime_DB.ChargerDelay_PT[i], ET => ChargeTime_DB.ChargerDelay_ET[i]);
						END_FOR;
						StartGLS3Charger := FALSE;
						ChargeTime_DB.PreFormChargeTime_TON (IN := FALSE, PT := ChargeTime_DB.PreFormChargeTime_PT, ET => ChargeTime_DB.PreFormChargeTime_ET);
						StartChargingBroadcast := FALSE; // reset the broadcast bit whne all chargers 
						ChargeTimeFinished := FALSE; //reset chargetime done bit
						ePulseState := E_PulseState.CHARGECOMPLETE;
					END_IF
	//Charge complete
	E_PulseState.CHARGECOMPLETE: 
	
					ChargeCompleted := FALSE; //reset bit
					ChargingRunOutTMR_TON (IN := FALSE);
					eStatus := E_Status.CHARGECOMPLETE;
					
					MCP_IO.GLS1_hvON := FALSE; //turn off spark gap charger
					MCP_IO.GLS2_hvON := FALSE;	
					SparkGapCharger_TON(IN := FALSE, PT := SparkGapCharger_PT, ET => SparkGapCharger_ET);
					//start run out timer
					ChargedRunOutTMR_TON (IN := TRUE, PT := HMI_DB.RunOutTMR_PT);
					
					IF ChargedRunOutTMR_TON.Q = TRUE THEN
						Trips_DB.ChargedTimerRunout := TRUE;
						ChargedRunOutTMR_TON (IN := FALSE, PT := HMI_DB.RunOutTMR_PT);
						ePulseState := E_PulseState.DUMPING;
					END_IF
					//turn off charger HV and inhibit 
					//FOR i := 1 TO 8 BY 1 DO 
					FOR i := 1 TO 3 BY 1 DO 
						MCP_IO.Charger[i].inhibit := TRUE;
						MCP_IO.Charger[i].HV_ON := FALSE; 
						ChargeTime_DB.ChargerDelay_TON[i] (IN := FALSE, PT := ChargeTime_DB.ChargerDelay_PT[i], ET => ChargeTime_DB.ChargerDelay_ET[i]);
					END_FOR
					MCP_IO.GLS3_hvON := FALSE;
					ChargeTime_DB.PreFormChargeTime_TON(IN := FALSE);
					
					IF eCommand = E_Command.DISCONNECT THEN 
						ePulseState := E_PulseState.DISCONNECTING;
					END_IF

	//Disconnecting
	E_PulseState.DISCONNECTING:
					eStatus := E_Status.DISCONNECTING;
					//setpoints to 0
					//FOR i := 1 TO 8 BY 1 DO
					FOR i := 1 TO 3 BY 1 DO
						MCP_IO.Charger[i].voltageSP := 0;
					END_FOR;
					MCP_IO.GLS3_voltageSP := 0;
					//spark gap chargers now turns off
					MCP_IO.GLS1_hvON := FALSE; 
					MCP_IO.GLS2_hvON := FALSE;
					MCP_IO.GLS1_voltageSP := 0;
					MCP_IO.GLS2_voltageSP := 0;
					
					//start run out timer
					ChargedRunOutTMR_TON (IN := TRUE, PT := HMI_DB.RunOutTMR_PT);
					
					IF ChargedRunOutTMR_TON.Q = TRUE THEN
						Trips_DB.ChargedTimerRunout := TRUE;
						ChargedRunOutTMR_TON (IN := FALSE, PT := HMI_DB.RunOutTMR_PT);
						ePulseState := E_PulseState.DUMPING;
					END_IF
					//keep dump relays open, 
					FOR j := 1 TO 3 BY 1 DO 
						//close all dump relays
						LCP.Section[j].Peak.OpenDumpRelay1 := TRUE;
						LCP.Section[j].Peak.OpenDumpRelay2 := TRUE;
						LCP.Section[j].Sust.OpenDumpRelay1 := TRUE;
						LCP.Section[j].Sust.OpenDumpRelay2 := TRUE;	
						//Open all charge relays
						LCP.Section[j].Peak.CloseChargeRelay1 := FALSE; 
						LCP.Section[j].Peak.CloseChargeRelay2 := FALSE; 
						LCP.Section[j].Sust.CloseChargeRelay1 := FALSE;
						LCP.Section[j].Sust.CloseChargeRelay2 := FALSE;
					END_FOR;	
					//close all dump relay on form
					LCP.Section[4].Form.OpenDumpRelay1 := TRUE;
					LCP.Section[4].Form.OpenDumpRelay2 := TRUE;
					LCP.Section[4].Form.OpenPreFormDumpRly := TRUE;
					LCP.Section[4].Form.OpenFormTrigDumpRly1 := TRUE;
					LCP.Section[4].Form.OpenPreFormTrigDumpRly1 := TRUE;

					//open all charge rly on form
					LCP.Section[4].Form.CloseChargeRelay1 := FALSE;
					LCP.Section[4].Form.CloseChargeRelay2 := FALSE;
					LCP.Section[4].Form.CloseFormTrigChargeRly := FALSE;
					LCP.Section[4].Form.ClosePreFormChargeRly := FALSE;
					LCP.Section[4].Form.ClosePreFormTrigChargeRly := FALSE;	
					
					IF Permissives_DB.AllChargeRelaysClosed = FALSE AND Permissives_DB.AllDumpRelaysOpen THEN
						eStatus := E_Status.DISCONNECTED; //send status to main plc
					END_IF;
					
					IF eCommand = E_Command.ABORT THEN 
						ePulseState := E_PulseState.ABORT;
					ELSIF eCommand = E_Command.DUMP THEN
						ePulseState := E_PulseState.DUMPING;
					END_IF;
	//Dumping
	E_PulseState.DUMPING:  
					//start dump runout timer
					DumpingRunOutTMR_TON (IN := TRUE, PT := DumpingRunOutTMR_PT, ET => DumpingRunOutTMR_ET);
					
					IF DumpingRunOutTMR_TON.Q = TRUE THEN //if timer run out, and in remoter mode go to trip
						Trips_DB.DumpTimerRunout := TRUE;
						DumpingRunOutTMR_TON (IN := FALSE);
						ePulseState := E_PulseState.TRIPPED;
					END_IF
					
					//TURN OFF ALL CHARGERS
					//FOR i := 1 TO 8 BY 1 DO 
					FOR i := 1 TO 3 BY 1 DO
						MCP_IO.Charger[i].inhibit := TRUE; 		
						MCP_IO.Charger[i].HV_ON := FALSE; 
						MCP_IO.Charger[i].voltageSP := 0;
			
						ChargeTime_DB.ChargingTimeElapse_TON[i] (IN := FALSE); //reset charging time elapse
					END_FOR;
					MCP_IO.GLS1_hvON := FALSE;
					MCP_IO.GLS2_hvON := FALSE;
					MCP_IO.GLS3_hvON := FALSE;
					MCP_IO.GLS1_voltageSP := 0;
					MCP_IO.GLS2_voltageSP := 0;
					MCP_IO.GLS3_voltageSP := 0;
					
					ChargeTime_DB.PreFormChargingTimeElapse_TON (IN := FALSE);
					//start delay
					AbortPSnRlyDelay_Timer (IN := TRUE, PT := AbortPSnRlyDelay_PT);					
					
					IF AbortPSnRlyDelay_Timer.Q = TRUE THEN 
						AbortPSnRlyDelayDONE := TRUE;
						AbortPSnRlyDelay_Timer (IN := FALSE);
					END_IF;
					
					IF 	AbortPSnRlyDelayDONE = TRUE THEN
						FOR j := 1 TO 3 BY 1 DO 
							//Open all charge relays
							LCP.Section[j].Peak.CloseChargeRelay1 := FALSE; 
							LCP.Section[j].Peak.CloseChargeRelay2 := FALSE; 
							LCP.Section[j].Sust.CloseChargeRelay1 := FALSE;
							LCP.Section[j].Sust.CloseChargeRelay2 := FALSE;
							//close all dump relays  - for SAFE STATE they can all go together
							LCP.Section[j].Peak.OpenDumpRelay1 := FALSE;
							LCP.Section[j].Peak.OpenDumpRelay2 := FALSE;
							LCP.Section[j].Sust.OpenDumpRelay1 := FALSE;
							LCP.Section[j].Sust.OpenDumpRelay2 := FALSE;	
						END_FOR;
						//open all charge rly on form
						LCP.Section[4].Form.CloseChargeRelay1 := FALSE;
						LCP.Section[4].Form.CloseChargeRelay2 := FALSE;
						LCP.Section[4].Form.CloseFormTrigChargeRly := FALSE;
						LCP.Section[4].Form.ClosePreFormChargeRly := FALSE;
						LCP.Section[4].Form.ClosePreFormTrigChargeRly := FALSE;
						//close all dump relay on form
						LCP.Section[4].Form.OpenDumpRelay1 := FALSE;
						LCP.Section[4].Form.OpenDumpRelay2 := FALSE;
						LCP.Section[4].Form.OpenPreFormDumpRly := FALSE;
						LCP.Section[4].Form.OpenFormTrigDumpRly1 := FALSE;
						LCP.Section[4].Form.OpenPreFormTrigDumpRly1 := FALSE;
						
						AbortPSnRlyDelay_Timer (IN := FALSE);
						AbortPSnRlyDelayDONE := FALSE;
					END_IF;
					
					eStatus := E_Status.DUMPING;
					
					IF (Permissives_DB.AllSectCapsDischarged = TRUE AND 
						Permissives_DB.AllDumpRelaysOpen = FALSE AND 
						eCommand = E_Command.IDLE AND 
						GVL.RemoteModeSelected = TRUE) 
						THEN 
							ePulseState := E_PulseState.SAFE;
					END_IF
	
	//Abort
	E_PulseState.ABORT: 
					//do something
					//ChargingRunOutTMR_TON (IN := FALSE);
					//TURN OFF ALL CHARGERS' outputs
					//FOR i := 1 TO 8 BY 1 DO
					FOR i := 1 TO 3 BY 1 DO 
						MCP_IO.Charger[i].inhibit := TRUE; //active low
						MCP_IO.Charger[i].HV_ON := FALSE; 
						MCP_IO.Charger[i].voltageSP := 0;
						
						ChargeTime_DB.ChargingTimeElapse_TON[i] (IN := FALSE);  
					END_FOR;
					MCP_IO.GLS1_hvON := FALSE;
					MCP_IO.GLS2_hvON := FALSE;
					MCP_IO.GLS3_hvON := FALSE;
					
					MCP_IO.GLS1_voltageSP := 0;
					MCP_IO.GLS2_voltageSP := 0;
					MCP_IO.GLS3_voltageSP := 0;
					//start delay
					AbortPSnRlyDelay_Timer (IN := TRUE, PT := AbortPSnRlyDelay_PT);					
					
					IF AbortPSnRlyDelay_Timer.Q = TRUE THEN 
						AbortPSnRlyDelayDONE := TRUE;
						AbortPSnRlyDelay_Timer (IN := FALSE);
					END_IF;
					IF AbortPSnRlyDelayDONE = TRUE THEN
						FOR j := 1 TO 3 BY 1 DO 
							//Open all charge relays
							LCP.Section[j].Peak.CloseChargeRelay1 := FALSE; 
							LCP.Section[j].Peak.CloseChargeRelay2 := FALSE; 
							LCP.Section[j].Sust.CloseChargeRelay1 := FALSE;
							LCP.Section[j].Sust.CloseChargeRelay2 := FALSE;
							//close all dump relays  - for SAFE STATE they can all go together
							LCP.Section[j].Peak.OpenDumpRelay1 := FALSE;
							LCP.Section[j].Peak.OpenDumpRelay2 := FALSE;
							LCP.Section[j].Sust.OpenDumpRelay1 := FALSE;
							LCP.Section[j].Sust.OpenDumpRelay2 := FALSE;	
						END_FOR;
						//open all charge rly on form
						LCP.Section[4].Form.CloseChargeRelay1 := FALSE;
						LCP.Section[4].Form.CloseChargeRelay2 := FALSE;
						LCP.Section[4].Form.CloseFormTrigChargeRly := FALSE;
						LCP.Section[4].Form.ClosePreFormChargeRly := FALSE;
						LCP.Section[4].Form.ClosePreFormTrigChargeRly := FALSE;
						//close all dump relay on form
						LCP.Section[4].Form.OpenDumpRelay1 := FALSE;
						LCP.Section[4].Form.OpenDumpRelay2 := FALSE;
						LCP.Section[4].Form.OpenPreFormDumpRly := FALSE;
						LCP.Section[4].Form.OpenFormTrigDumpRly1 := FALSE;
						LCP.Section[4].Form.OpenPreFormTrigDumpRly1 := FALSE;
						
						AbortPSnRlyDelay_Timer (IN := FALSE);
						AbortPSnRlyDelayDONE := FALSE;		
					END_IF;
	
					eStatus := E_Status.ABORT;
					//logic to go back to safe state.
					IF (Trips_DB.NoFaultDetected = TRUE AND 
						Permissives_DB.AllDumpRelaysOpen = FALSE AND 
						Permissives_DB.AllChargeRelaysClosed = FALSE AND
						Permissives_DB.AllChargerHVisON = FALSE) OR (eCommand = E_Command.IDLE AND MCP_IO.RemoteModeSelected = TRUE)
						THEN 
							AbortPSnRlyDelayDONE := FALSE;
							ePulseState := E_PulseState.SAFE;	
					END_IF;
					
	//Abort
	E_PulseState.TRIPPED: 
					eStatus := E_Status.TRIPPED;
					//reset dumping run out timer
					DumpingRunOutTMR_TON (IN := FALSE, PT := DumpingRunOutTMR_PT, ET => DumpingRunOutTMR_ET);
					
					//FOR i := 1 TO 8 BY 1 DO
					FOR i := 1 TO 3 BY 1 DO 
						MCP_IO.Charger[i].inhibit := TRUE; //active low
						MCP_IO.Charger[i].HV_ON := FALSE; 
					END_FOR;
					
					FOR j := 1 TO 3 BY 1 DO 
						//close all dump relays
						LCP.Section[j].Peak.OpenDumpRelay1 := FALSE;
						LCP.Section[j].Peak.OpenDumpRelay2 := FALSE;
						LCP.Section[j].Sust.OpenDumpRelay1 := FALSE;
						LCP.Section[j].Sust.OpenDumpRelay2 := FALSE;
						//Open all charge relays
						LCP.Section[j].Peak.CloseChargeRelay1 := FALSE; 
						LCP.Section[j].Peak.CloseChargeRelay2 := FALSE; 
						LCP.Section[j].Sust.CloseChargeRelay1 := FALSE;
						LCP.Section[j].Sust.CloseChargeRelay2 := FALSE;	
					END_FOR;	
					//close all dump relay on form
					LCP.Section[4].Form.OpenDumpRelay1 := FALSE;
					LCP.Section[4].Form.OpenDumpRelay2 := FALSE;
					LCP.Section[4].Form.OpenPreFormDumpRly := FALSE;
					LCP.Section[4].Form.OpenFormTrigDumpRly1 := FALSE;
					LCP.Section[4].Form.OpenPreFormTrigDumpRly1 := FALSE;
			
					//open all charge rly on form
					LCP.Section[4].Form.CloseChargeRelay1 := FALSE;
					LCP.Section[4].Form.CloseChargeRelay2 := FALSE;
					LCP.Section[4].Form.CloseFormTrigChargeRly := FALSE;
					LCP.Section[4].Form.ClosePreFormChargeRly := FALSE;
					LCP.Section[4].Form.ClosePreFormTrigChargeRly := FALSE;	
	
					//FOR i := 1 TO 8 BY 1 DO
					FOR i := 1 TO 3 BY 1 DO
						MCP_IO.Charger[i].voltageSP := 0;
						ChargeTime_DB.ChargingTimeElapse_TON[i] (IN := FALSE);  
					END_FOR;					
					MCP_IO.GLS1_hvON := FALSE;
					MCP_IO.GLS2_hvON := FALSE;
					MCP_IO.GLS3_hvON := FALSE;
					
					MCP_IO.GLS1_voltageSP := 0;
					MCP_IO.GLS2_voltageSP := 0;
					MCP_IO.GLS3_voltageSP := 0;
									
					//ChargingRunOutTMR_TON (IN := FALSE);
					//logic to go back to safe state.
					IF (Trips_DB.NoFaultDetected = TRUE OR HMI_DB.NoFaultDetectedBP = TRUE) AND 
						(Permissives_DB.AllDumpRelaysOpen = FALSE OR HMI_DB.AllDumpRelaysOpenBP = TRUE) AND 
						(Permissives_DB.AllChargeRelaysClosed = FALSE OR HMI_DB.AllChargeRelayCloseBP = TRUE) AND
						Permissives_DB.AllChargerHVisON = FALSE  AND
						(Permissives_DB.SafetyOK = TRUE OR HMI_DB.SafetyOKBP = TRUE)
						THEN 
							ePulseState := E_PulseState.SAFE;	
					END_IF;
	//lOCAL MODE
	E_PulseState.LOCALMODE:
					eStatus := E_Status.LOCAL_MODE;
					
					IF HMI_DB.DumpALLPB_Local = TRUE THEN
						LocalDumpActive := TRUE;
					END_IF
					
					//Local dump activated			
					IF LocalDumpActive = TRUE THEN 
						//reset all HMI Switches
						HMI_DB.OpenAllDumpRlyPB := FALSE;
						HMI_DB.CloseAllChargeRlyPB := FALSE;
						
						HMI_DB.CloseAllPeakChargRlySW := FALSE;
						HMI_DB.CloseAllSustChargRlySW := FALSE;
						HMI_DB.CloseAllFormChargRlySW := FALSE;
						HMI_DB.CloseAllPreFormChargRlySW := FALSE;
						HMI_DB.ClosePreFormTrigChargeRlySW := FALSE;
						HMI_DB.CloseFormTrigChargeRlySW := FALSE;
						
						HMI_DB.OpenAllPeakDumpRlySW := FALSE;
						HMI_DB.OpenAllSustDumpRlySW := FALSE;
						HMI_DB.OpenAllFormDumpRlySW := FALSE;
						HMI_DB.OpenAllPreFormDumpRlySW := FALSE;
						HMI_DB.OpenPreFormTrigDumpRlySW := FALSE;
						HMI_DB.OpenFormTrigDumpRlySW := FALSE;
						
						HMI_DB.PeakHVONsw := FALSE;
						HMI_DB.SustHVONsw := FALSE;
						HMI_DB.FormHVONsw := FALSE;
						HMI_DB.PreFormHVONsw := FALSE;
						HMI_DB.GLS1HVONsw := FALSE;
						HMI_DB.GLS2HVONsw := FALSE;			
						
						Dump( EN := TRUE, IN1 := Permissives_DB.AllSectCapsDischarged, IN2 := Permissives_DB.AllDumpRelaysOpen);
						DumpingRunOutTMR_TON (IN := TRUE, PT := DumpingRunOutTMR_PT, ET => DumpingRunOutTMR_ET);
						LocalDumpElapse := Dump.DumpingRunOut_Elapse;
						ELSE 
							Dump.EN := FALSE; 
							DumpingRunOutTMR_TON (IN := FALSE);
					END_IF;
					
					IF DumpingRunOutTMR_TON.Q = TRUE THEN 
						Trips_DB.DumpTimerRunout := TRUE;
						DumpingRunOutTMR_TON (IN := FALSE);
					END_IF
					
					IF Trips_DB.DumpTimerRunout = TRUE THEN
						ePulseState := E_PulseState.TRIPPED;
					END_IF

 					IF Dump.DONE = TRUE THEN 
						LocalDumpActive := FALSE;
						Dump.EN := FALSE; 
						DumpingRunOutTMR_TON (IN := FALSE);
					END_IF
					//ChargingRunOutTMR_TON (IN := FALSE);
				//Start up procedure run*******************************************	
					//HMI Input TO Charger SP
					IF HMI_DB.PeakChargerSP > 10 THEN
						HMI_DB.PeakChargerSP := 10;
						ELSIF HMI_DB.PeakChargerSP <= 0 THEN
							HMI_DB.PeakChargerSP := 0;
					END_IF
					IF HMI_DB.SustChargerSP > 10 THEN 
						HMI_DB.SustChargerSP := 10;
						ELSIF HMI_DB.SustChargerSP <= 0 THEN
							HMI_DB.SustChargerSP := 0;
					END_IF
					IF HMI_DB.FormChargerSP > 35 THEN 
						HMI_DB.FormChargerSP := 35;
						ELSIF HMI_DB.FormChargerSP <= 0 THEN
							HMI_DB.FormChargerSP := 0;
					END_IF	
					IF HMI_DB.PreFormChargerSP > 30 THEN 
						HMI_DB.PreFormChargerSP := 30;
						ELSIF HMI_DB.PreFormChargerSP <= 0 THEN
							HMI_DB.PreFormChargerSP := 0;
					END_IF	
					IF HMI_DB.FormTrigChargerSP > 50 THEN 
						HMI_DB.FormTrigChargerSP := 50;
						ELSIF HMI_DB.FormTrigChargerSP <= 0 THEN
							HMI_DB.FormTrigChargerSP := 0;
					END_IF	
					IF HMI_DB.PreFormTrigChargerSP > 30 THEN 
						HMI_DB.PreFormTrigChargerSP := 30;
						ELSIF HMI_DB.PreFormTrigChargerSP <= 0 THEN
							HMI_DB.PreFormTrigChargerSP := 0;
					END_IF				
					//char 1 - 3 is peaking, 4 - 6 sust, 7 - 8 form, gls 3 is preform
					MCP_IO.Charger[1].voltageSP := HMI_DB.PeakChargerSP * 1000;
					MCP_IO.Charger[2].voltageSP := HMI_DB.PeakChargerSP * 1000;
					MCP_IO.Charger[3].voltageSP := HMI_DB.PeakChargerSP * 1000;
					(*MCP_IO.Charger[4].voltageSP := HMI_DB.SustChargerSP * 1000;
					MCP_IO.Charger[5].voltageSP := HMI_DB.SustChargerSP * 1000;
					MCP_IO.Charger[6].voltageSP := HMI_DB.SustChargerSP * 1000;			
					MCP_IO.Charger[7].voltageSP := HMI_DB.FormChargerSP * 1000;
					MCP_IO.Charger[8].voltageSP := HMI_DB.FormChargerSP * 1000;	*)
					MCP_IO.GLS3_voltageSP := HMI_DB.PreFormChargerSP * 1000;
					MCP_IO.GLS1_voltageSP := HMI_DB.FormTrigChargerSP * 1000;
					MCP_IO.GLS2_voltageSP := HMI_DB.PreFormTrigChargerSP * 1000;
					
					IF HMI_DB.CloseAllChargeRlyPB = TRUE AND Trips_DB.NoFaultDetected = TRUE AND Permissives_DB.AllChargerHVisON = FALSE AND Permissives_DB.AllChargerInhibited = TRUE THEN
						FOR j := 1 TO 3 BY 1 DO 
							//CLOSE all charge relays
							LCP.Section[j].Peak.CloseChargeRelay1 := TRUE; 
							LCP.Section[j].Peak.CloseChargeRelay2 := TRUE; 
							LCP.Section[j].Sust.CloseChargeRelay1 := TRUE;
							LCP.Section[j].Sust.CloseChargeRelay2 := TRUE;
						END_FOR;
						//CLOSE all charge rly on form
						LCP.Section[4].Form.CloseChargeRelay1 := TRUE;
						LCP.Section[4].Form.CloseChargeRelay2 := TRUE;
						LCP.Section[4].Form.CloseFormTrigChargeRly := TRUE;
						LCP.Section[4].Form.ClosePreFormChargeRly := TRUE;
						LCP.Section[4].Form.ClosePreFormTrigChargeRly := TRUE;
					ELSE
						FOR j := 1 TO 3 BY 1 DO 
							//Open all charge relays
							LCP.Section[j].Peak.CloseChargeRelay1 := FALSE; 
							LCP.Section[j].Peak.CloseChargeRelay2 := FALSE; 
							LCP.Section[j].Sust.CloseChargeRelay1 := FALSE;
							LCP.Section[j].Sust.CloseChargeRelay2 := FALSE;
						END_FOR;
						//open all charge rly on form
						LCP.Section[4].Form.CloseChargeRelay1 := FALSE;
						LCP.Section[4].Form.CloseChargeRelay2 := FALSE;
						LCP.Section[4].Form.CloseFormTrigChargeRly := FALSE;
						LCP.Section[4].Form.ClosePreFormChargeRly := FALSE;
						LCP.Section[4].Form.ClosePreFormTrigChargeRly := FALSE;	
					END_IF;
					
					//OPEN DUMP
					IF HMI_DB.OpenAllDumpRlyPB = TRUE AND Trips_DB.NoFaultDetected = TRUE AND Permissives_DB.AllChargerHVisON = FALSE AND Permissives_DB.AllChargerInhibited = TRUE THEN
						FOR j := 1 TO 3 BY 1 DO 
							//open all dump relays  - for SAFE STATE they can all go together
							LCP.Section[j].Peak.OpenDumpRelay1 := TRUE;
							LCP.Section[j].Peak.OpenDumpRelay2 := TRUE;
							LCP.Section[j].Sust.OpenDumpRelay1 := TRUE;
							LCP.Section[j].Sust.OpenDumpRelay2 := TRUE;	
						END_FOR;	
						//close all dump relay on form
						LCP.Section[4].Form.OpenDumpRelay1 := TRUE;
						LCP.Section[4].Form.OpenDumpRelay2 := TRUE;
						LCP.Section[4].Form.OpenPreFormDumpRly := TRUE;
						LCP.Section[4].Form.OpenFormTrigDumpRly1 := TRUE;
						LCP.Section[4].Form.OpenPreFormTrigDumpRly1 := TRUE;					
					ELSE
						FOR j := 1 TO 3 BY 1 DO 
							//open all dump relays  - for SAFE STATE they can all go together
							LCP.Section[j].Peak.OpenDumpRelay1 := FALSE;
							LCP.Section[j].Peak.OpenDumpRelay2 := FALSE;
							LCP.Section[j].Sust.OpenDumpRelay1 := FALSE;
							LCP.Section[j].Sust.OpenDumpRelay2 := FALSE;	
						END_FOR;	
						//close all dump relay on form
						LCP.Section[4].Form.OpenDumpRelay1 := FALSE;
						LCP.Section[4].Form.OpenDumpRelay2 := FALSE;
						LCP.Section[4].Form.OpenPreFormDumpRly := FALSE;
						LCP.Section[4].Form.OpenFormTrigDumpRly1 := FALSE;
						LCP.Section[4].Form.OpenPreFormTrigDumpRly1 := FALSE;	
					END_IF;
					
					IF HMI_DB.LiftMachineGNDsw = TRUE AND Trips_DB.NoFaultDetected = TRUE THEN
						MCP_IO.LiftMachineGND := TRUE;
						ELSE
							MCP_IO.LiftMachineGND := FALSE;
					END_IF;
					// no fault, safety ok, charger HV is OFF and Inhibited condition before opening dump relays
					IF Trips_DB.NoFaultDetected = TRUE AND 
						Permissives_DB.SafetyOK = TRUE AND
						Permissives_DB.AllPeakChargerHVisON = FALSE AND 
						Permissives_DB.AllPeakChargerInhibited = TRUE AND 
						HMI_DB.OpenAllPeakDumpRlySW = TRUE 
						THEN
							FOR j := 1 TO 3 BY 1 DO 
								//open all peak dump relays 
								LCP.Section[j].Peak.OpenDumpRelay1 := TRUE;
								LCP.Section[j].Peak.OpenDumpRelay2 := TRUE;	
							END_FOR;
						ELSIF HMI_DB.OpenAllPeakDumpRlySW = FALSE THEN
								FOR j := 1 TO 3 BY 1 DO 
									LCP.Section[j].Peak.OpenDumpRelay1 := FALSE;
									LCP.Section[j].Peak.OpenDumpRelay2 := FALSE;	
								END_FOR;
					END_IF

					IF Trips_DB.NoFaultDetected = TRUE AND 
						Permissives_DB.SafetyOK = TRUE AND
						Permissives_DB.AllSustChargerHVisON = FALSE AND 
						Permissives_DB.AllSustChargerInhibited = TRUE AND 
						HMI_DB.OpenAllSustDumpRlySW = TRUE 
						THEN
							FOR j := 1 TO 3 BY 1 DO 
								//open all sust dump relays 
								LCP.Section[j].Sust.OpenDumpRelay1 := TRUE;
								LCP.Section[j].Sust.OpenDumpRelay2 := TRUE;	
							END_FOR;
						ELSIF HMI_DB.OpenAllSustDumpRlySW = FALSE THEN 
								FOR j := 1 TO 3 BY 1 DO 
									LCP.Section[j].Sust.OpenDumpRelay1 := FALSE;
									LCP.Section[j].Sust.OpenDumpRelay2 := FALSE;	
								END_FOR;							
					END_IF
					
					IF Trips_DB.NoFaultDetected = TRUE AND 
						Permissives_DB.SafetyOK = TRUE AND
						Permissives_DB.AllFormChargerHVisON = FALSE AND 
						Permissives_DB.AllFormChargerInhibited = TRUE AND 
						HMI_DB.OpenAllFormDumpRlySW = TRUE 
						THEN
							//open all form dump relays 
							LCP.Section[4].Form.OpenDumpRelay1 := TRUE;
							LCP.Section[4].Form.OpenDumpRelay2 := TRUE;	
						ELSIF HMI_DB.OpenAllFormDumpRlySW = FALSE THEN 
								LCP.Section[4].Form.OpenDumpRelay1 := FALSE;
								LCP.Section[4].Form.OpenDumpRelay2 := FALSE;								
					END_IF					
					// preform dump
					IF Trips_DB.NoFaultDetected = TRUE AND 
						Permissives_DB.SafetyOK = TRUE AND
						LCP.Section[4].Form.PreFormChargeRly_close = FALSE AND //charge relays open
						HMI_DB.OpenAllPreFormDumpRlySW = TRUE 
						THEN
							//OPEN ALL preform dump relay
							LCP.Section[4].Form.OpenPreFormDumpRly := TRUE;
						ELSIF HMI_DB.OpenAllPreFormDumpRlySW = FALSE THEN  
								LCP.Section[4].Form.OpenPreFormDumpRly := FALSE;
					END_IF;
					
					//preform trig dump 
					IF Trips_DB.NoFaultDetected = TRUE AND 
						Permissives_DB.SafetyOK = TRUE AND
						LCP.Section[4].Form.PreFormTrigChargeRly_close = FALSE AND //charge relays open
						HMI_DB.OpenPreFormTrigDumpRlySW = TRUE 
						THEN
							//OPEN ALL preform trig dump relay
							LCP.Section[4].Form.OpenPreFormTrigDumpRly1 := TRUE;
						ELSIF HMI_DB.OpenPreFormTrigDumpRlySW = FALSE THEN
								LCP.Section[4].Form.OpenPreFormTrigDumpRly1 := FALSE;
					END_IF;					
					//form  trig dump 
					IF Trips_DB.NoFaultDetected = TRUE AND 
						Permissives_DB.SafetyOK = TRUE AND
						LCP.Section[4].Form.FormTrigChargeRly_close = FALSE AND //charge relays open
						HMI_DB.OpenFormTrigDumpRlySW = TRUE 
						THEN					
							LCP.Section[4].Form.OpenFormTrigDumpRly1 := TRUE;
						ELSIF HMI_DB.OpenFormTrigDumpRlySW = FALSE THEN
							LCP.Section[4].Form.OpenFormTrigDumpRly1 := FALSE;
					END_IF;
					
					//Charge relays
					//peak charge 
					IF Trips_DB.NoFaultDetected = TRUE AND 
						Permissives_DB.SafetyOK = TRUE AND
						Permissives_DB.AllPeakChargerHVisON = FALSE AND 
						Permissives_DB.AllPeakChargerInhibited = TRUE AND 
						Permissives_DB.AllPeakDumpRlyOpen = TRUE AND 
						HMI_DB.CloseAllPeakChargRlySW = TRUE
						THEN
							LCP.Section[1].Peak.CloseChargeRelay1 := TRUE;
							LCP.Section[1].Peak.CloseChargeRelay2 := TRUE;
							LCP.Section[2].Peak.CloseChargeRelay1 := TRUE;
							LCP.Section[2].Peak.CloseChargeRelay2 := TRUE;
							LCP.Section[3].Peak.CloseChargeRelay1 := TRUE;
							LCP.Section[3].Peak.CloseChargeRelay2 := TRUE;
						ELSIF Permissives_DB.AllPeakChargerHVisON = FALSE AND Permissives_DB.AllPeakChargerInhibited = TRUE AND HMI_DB.CloseAllPeakChargRlySW = FALSE 
							THEN
								LCP.Section[1].Peak.CloseChargeRelay1 := FALSE;
								LCP.Section[1].Peak.CloseChargeRelay2 := FALSE;
								LCP.Section[2].Peak.CloseChargeRelay1 := FALSE;
								LCP.Section[2].Peak.CloseChargeRelay2 := FALSE;
								LCP.Section[3].Peak.CloseChargeRelay1 := FALSE;
								LCP.Section[3].Peak.CloseChargeRelay2 := FALSE;
					END_IF;
					
					//sust charge
					IF Trips_DB.NoFaultDetected = TRUE AND 
						Permissives_DB.SafetyOK = TRUE AND
						Permissives_DB.AllSustChargerHVisON = FALSE AND 
						Permissives_DB.AllSustChargerInhibited = TRUE AND 
						Permissives_DB.AllSustDumpRlyOpen = TRUE AND 
						HMI_DB.CloseAllSustChargRlySW = TRUE
						THEN
							LCP.Section[1].Sust.CloseChargeRelay1 := TRUE;
							LCP.Section[1].Sust.CloseChargeRelay2 := TRUE;
							LCP.Section[2].Sust.CloseChargeRelay1 := TRUE;
							LCP.Section[2].Sust.CloseChargeRelay2 := TRUE;
							LCP.Section[3].Sust.CloseChargeRelay1 := TRUE;
							LCP.Section[3].Sust.CloseChargeRelay2 := TRUE;
						ELSIF Permissives_DB.AllSustChargerHVisON = FALSE AND Permissives_DB.AllSustChargerInhibited = TRUE AND HMI_DB.CloseAllSustChargRlySW = FALSE 
							THEN
								LCP.Section[1].Sust.CloseChargeRelay1 := FALSE;
								LCP.Section[1].Sust.CloseChargeRelay2 := FALSE;
								LCP.Section[2].Sust.CloseChargeRelay1 := FALSE;
								LCP.Section[2].Sust.CloseChargeRelay2 := FALSE;
								LCP.Section[3].Sust.CloseChargeRelay1 := FALSE;
								LCP.Section[3].Sust.CloseChargeRelay2 := FALSE;
					END_IF;
					
					//Form charge
					IF Trips_DB.NoFaultDetected = TRUE AND 
						Permissives_DB.SafetyOK = TRUE AND
						Permissives_DB.AllFormChargerHVisON = FALSE AND 
						Permissives_DB.AllFormChargerInhibited = TRUE AND 
						Permissives_DB.AllFormDumpRlyOpen = TRUE AND 
						HMI_DB.CloseAllFormChargRlySW = TRUE
						THEN
							LCP.Section[4].Form.CloseChargeRelay1 := TRUE;
							LCP.Section[4].Form.CloseChargeRelay2 := TRUE;
						ELSIF Permissives_DB.AllFormChargerHVisON = FALSE AND Permissives_DB.AllFormChargerInhibited = TRUE AND HMI_DB.CloseAllFormChargRlySW = FALSE 
							THEN
								LCP.Section[4].Form.CloseChargeRelay1 := TRUE;
								LCP.Section[4].Form.CloseChargeRelay2 := TRUE;
					END_IF;
					
					//preform charge - gls 3
					IF Trips_DB.NoFaultDetected = TRUE AND 
						Permissives_DB.SafetyOK = TRUE AND
						MCP_IO.GLS3_hvON = FALSE AND  
						LCP.Section[4].Form.PreFormDumpRly_close = FALSE AND 
						HMI_DB.CloseAllPreFormChargRlySW = TRUE
						THEN 
							LCP.Section[4].Form.ClosePreFormChargeRly := TRUE;
						ELSIF MCP_IO.GLS3_hvON = FALSE AND HMI_DB.CloseAllPreFormChargRlySW = FALSE
							THEN
								LCP.Section[4].Form.ClosePreFormChargeRly := FALSE;
					END_IF;
					
					//preform trig charg - GLS 2
					IF Trips_DB.NoFaultDetected = TRUE AND 
						Permissives_DB.SafetyOK = TRUE AND
						MCP_IO.GLS2_hvON = FALSE AND  
						LCP.Section[4].Form.PreFormTrigDumpRly1_close = FALSE AND 
						HMI_DB.ClosePreFormTrigChargeRlySW = TRUE
						THEN 
							LCP.Section[4].Form.ClosePreFormTrigChargeRly := TRUE;
						ELSIF MCP_IO.GLS1_hvON = FALSE AND HMI_DB.ClosePreFormTrigChargeRlySW = FALSE
							THEN
								LCP.Section[4].Form.ClosePreFormTrigChargeRly := FALSE;
					END_IF;	
					
					//form trig charg - GLS 1
					IF Trips_DB.NoFaultDetected = TRUE AND 
						Permissives_DB.SafetyOK = TRUE AND
						MCP_IO.GLS1_hvON = FALSE AND 
						LCP.Section[4].Form.FormTrigDumpRly1_close = FALSE AND 
						HMI_DB.CloseFormTrigChargeRlySW = TRUE
						THEN 
							LCP.Section[4].Form.CloseFormTrigChargeRly := TRUE;
						ELSIF MCP_IO.GLS1_hvON = FALSE AND HMI_DB.CloseFormTrigChargeRlySW = FALSE
							THEN
								LCP.Section[4].Form.CloseFormTrigChargeRly := FALSE;
					END_IF;										
					//hv enable 
					//peak
					IF Trips_DB.NoFaultDetected = TRUE AND
						Permissives_DB.SafetyOK = TRUE AND 
						Permissives_DB.AllPeakChargeRlyClose = TRUE AND 
						Permissives_DB.AllPeakDumpRlyOpen = TRUE AND 
						HMI_DB.PeakHVONsw = TRUE 
						THEN 
							MCP_IO.Charger[1].HV_ON := TRUE;
							MCP_IO.Charger[1].inhibit := FALSE;
							MCP_IO.Charger[2].HV_ON := TRUE;
							MCP_IO.Charger[2].inhibit := FALSE;
							MCP_IO.Charger[3].HV_ON := TRUE;
							MCP_IO.Charger[3].inhibit := FALSE;
						ELSE
							MCP_IO.Charger[1].HV_ON := FALSE;
							MCP_IO.Charger[1].inhibit := TRUE;
							MCP_IO.Charger[2].HV_ON := FALSE;
							MCP_IO.Charger[2].inhibit := TRUE;
							MCP_IO.Charger[3].HV_ON := FALSE;
							MCP_IO.Charger[3].inhibit := TRUE;
					END_IF
					
					//sust
					(*IF Trips_DB.NoFaultDetected = TRUE AND
						Permissives_DB.SafetyOK = TRUE AND 
						Permissives_DB.AllSustChargeRlyClose = TRUE AND 
						Permissives_DB.AllSustDumpRlyOpen = TRUE AND 
						HMI_DB.SustHVONsw = TRUE 
						THEN 
							MCP_IO.Charger[4].HV_ON := TRUE;
							MCP_IO.Charger[4].inhibit := FALSE;
							MCP_IO.Charger[5].HV_ON := TRUE;
							MCP_IO.Charger[5].inhibit := FALSE;
							MCP_IO.Charger[6].HV_ON := TRUE;
							MCP_IO.Charger[6].inhibit := FALSE;
						ELSE
							MCP_IO.Charger[4].HV_ON := FALSE;
							MCP_IO.Charger[4].inhibit := TRUE;
							MCP_IO.Charger[5].HV_ON := FALSE;
							MCP_IO.Charger[5].inhibit := TRUE;
							MCP_IO.Charger[6].HV_ON := FALSE;
							MCP_IO.Charger[6].inhibit := TRUE;
					END_IF*)
					
					//Form
					(*IF Trips_DB.NoFaultDetected = TRUE AND
						Permissives_DB.SafetyOK = TRUE AND 
						Permissives_DB.AllFormChargeRlyClose = TRUE AND 
						Permissives_DB.AllFormDumpRlyOpen = TRUE AND 
						HMI_DB.FormHVONsw = TRUE 
						THEN 
							MCP_IO.Charger[7].HV_ON := TRUE;
							MCP_IO.Charger[7].inhibit := FALSE;
							MCP_IO.Charger[8].HV_ON := TRUE;
							MCP_IO.Charger[8].inhibit := FALSE;
						ELSE
							MCP_IO.Charger[7].HV_ON := FALSE;
							MCP_IO.Charger[7].inhibit := TRUE;
							MCP_IO.Charger[8].HV_ON := FALSE;
							MCP_IO.Charger[8].inhibit := TRUE;
					END_IF*)
					
					//preform
					IF Trips_DB.NoFaultDetected = TRUE AND
						Permissives_DB.SafetyOK = TRUE AND 
						LCP.Section[4].Form.PreFormChargeRly_close = TRUE AND 
						LCP.Section[4].Form.PreFormDumpRly_close = FALSE AND 
						HMI_DB.PreFormHVONsw = TRUE 
						THEN 
							MCP_IO.GLS3_hvON := TRUE;
						ELSE
							MCP_IO.GLS3_hvON := FALSE;			
					END_IF
					
					//preform trig
					IF Trips_DB.NoFaultDetected = TRUE AND
						Permissives_DB.SafetyOK = TRUE AND 
						LCP.Section[4].Form.PreFormTrigChargeRly_close = TRUE AND 
						LCP.Section[4].Form.PreFormTrigDumpRly1_close = FALSE AND 
						HMI_DB.GLS2HVONsw = TRUE 
						THEN 
							MCP_IO.GLS2_hvON := TRUE;
						ELSE
							MCP_IO.GLS2_hvON := FALSE;			
					END_IF	
					
					//form trig
					IF Trips_DB.NoFaultDetected = TRUE AND
						Permissives_DB.SafetyOK = TRUE AND 
						LCP.Section[4].Form.FormTrigChargeRly_close = TRUE AND 
						LCP.Section[4].Form.FormTrigDumpRly1_close = FALSE AND 
						HMI_DB.GLS1HVONsw = TRUE 
						THEN 
							MCP_IO.GLS1_hvON := TRUE;
						ELSE
							MCP_IO.GLS1_hvON := FALSE;			
					END_IF	
					
					IF GVL.RemoteModeSelected = TRUE THEN 
						ePulseState := E_PulseState.SAFE;
					END_IF
END_CASE;


//IF i > 8 THEN
IF i > 3 THEN
	i := 1;
END_IF

IF j > 3 THEN
	j := 1;
END_IF

//IF k > 8 THEN
IF k > 3 THEN
	k := 1;
END_IF

END_PROGRAM
